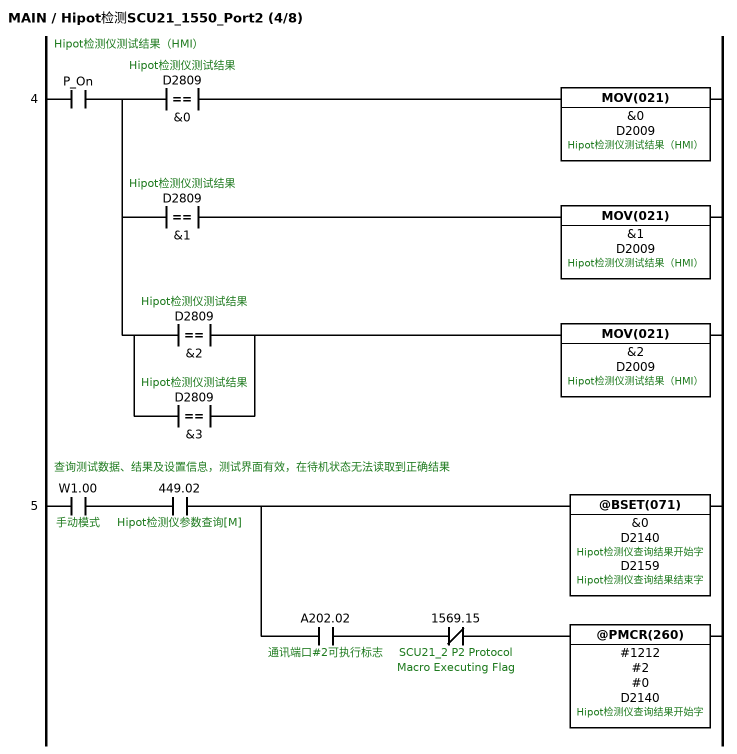
; [picture p48: MAIN / Hipot检测SCU21_1550_Port2, rungs 4-5]
; rung 4: Hipot检测仪测试结果（HMI）
LD P_On
OUT TR0
AND=(300) D2809 &0  ; Hipot检测仪测试结果
MOV(021) &0 D2009  ; Hipot检测仪测试结果（HMI）  // 0=无测试
LD TR0
AND=(300) D2809 &1  ; Hipot检测仪测试结果
MOV(021) &1 D2009  ; Hipot检测仪测试结果（HMI）  // 1=OK
LD TR0
LD=(300) D2809 &2  ; Hipot检测仪测试结果
OR=(300) D2809 &3  ; Hipot检测仪测试结果
ANDLD
MOV(021) &2 D2009  ; Hipot检测仪测试结果（HMI）  // 2=NG
; rung 5: 查询测试数据、结果及设置信息，测试界面有效，在待机状态无法读取到正确结果
LD W1.00  ; 手动模式
AND 449.02  ; Hipot检测仪参数查询[M]
@BSET(071) &0 D2140 D2159  ; Hipot检测仪查询结果开始字, Hipot检测仪查询结果结束字
AND A202.02  ; 通讯端口#2可执行标志
ANDNOT 1569.15  ; SCU21_2 P2 Protocol Macro Executing Flag
@PMCR(260) #1212 #2 #0 D2140  ; Hipot检测仪查询结果开始字

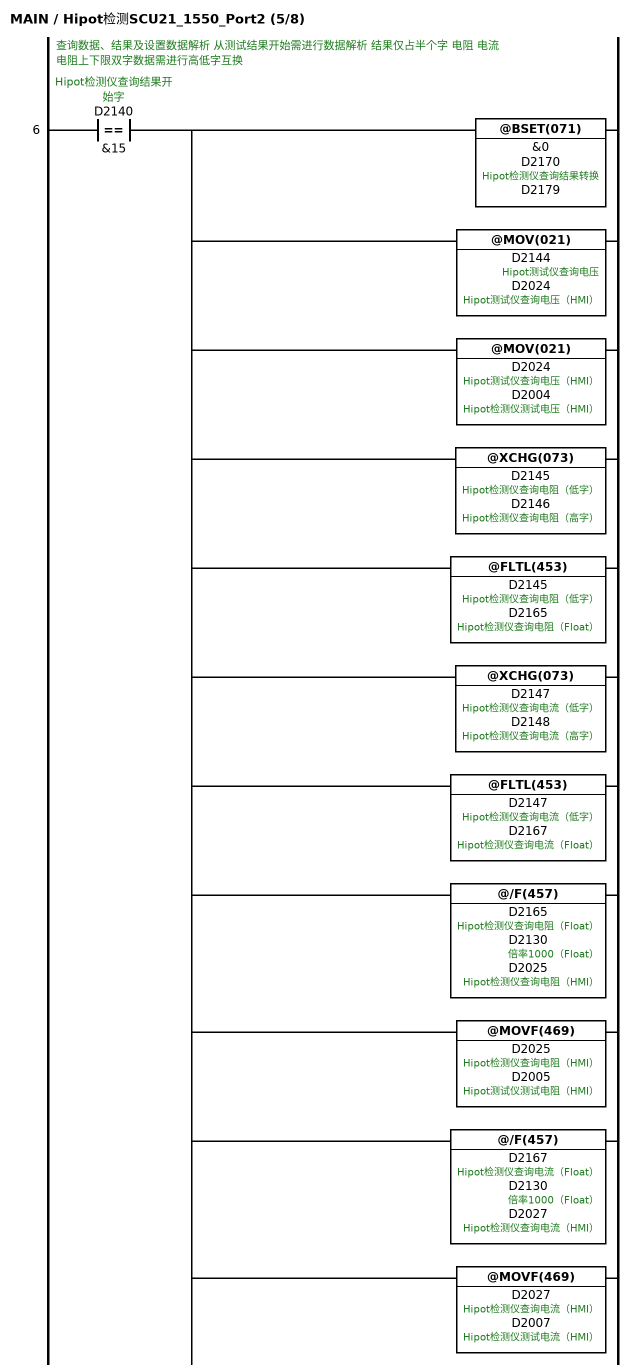

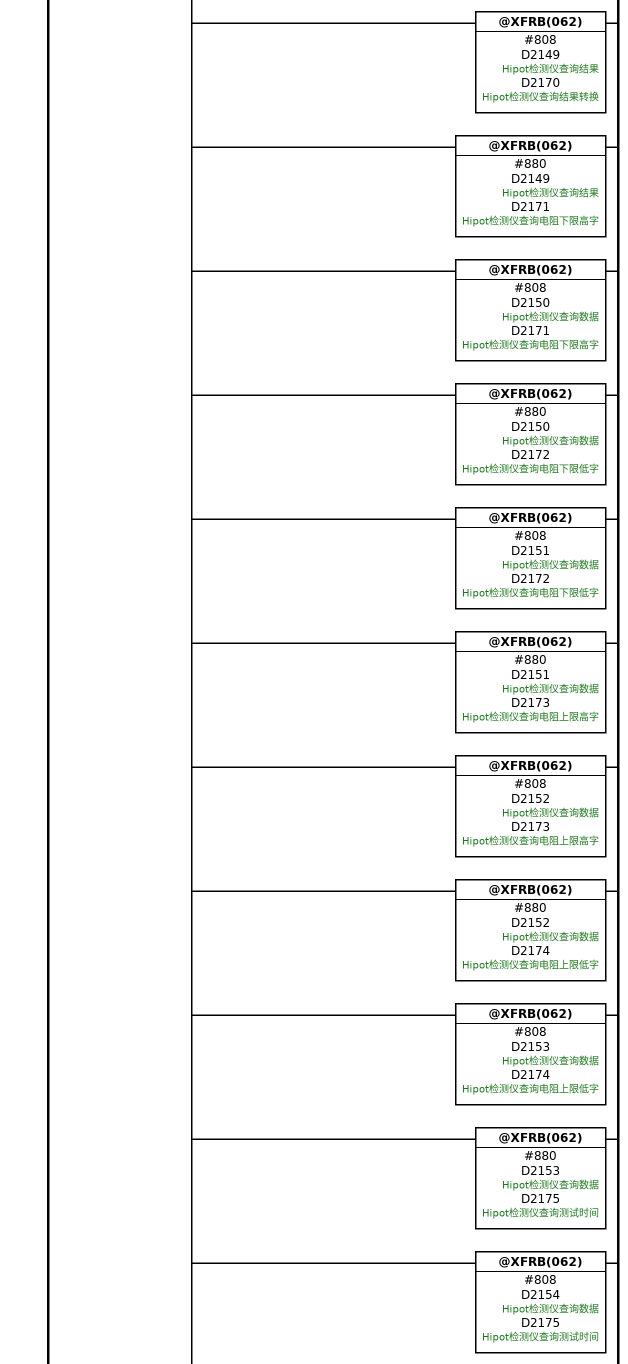

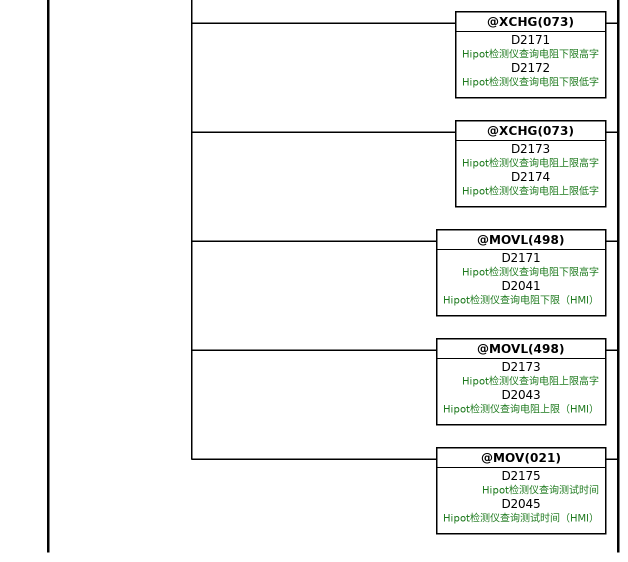
; rung 6: 查询数据、结果及设置数据解析 从测试结果开始需进行数据解析 结果仅占半个字 电阻 电流 电阻上下限双字数据需进行高低字互换
LD=(300) D2140 &15  ; Hipot检测仪查询结果开始字
@BSET(071) &0 D2170 D2179  ; Hipot检测仪查询结果转换
@MOV(021) D2144 D2024  ; Hipot测试仪查询电压, Hipot测试仪查询电压（HMI）
@MOV(021) D2024 D2004  ; Hipot测试仪查询电压（HMI）, Hipot检测仪测试电压（HMI）
@XCHG(073) D2145 D2146  ; Hipot检测仪查询电阻（低字）, Hipot检测仪查询电阻（高字）
@FLTL(453) D2145 D2165  ; Hipot检测仪查询电阻（低字）, Hipot检测仪查询电阻（Float）
@XCHG(073) D2147 D2148  ; Hipot检测仪查询电流（低字）, Hipot检测仪查询电流（高字）
@FLTL(453) D2147 D2167  ; Hipot检测仪查询电流（低字）, Hipot检测仪查询电流（Float）
@/F(457) D2165 D2130 D2025  ; Hipot检测仪查询电阻（Float）, 倍率1000（Float）, Hipot检测仪查询电阻（HMI）  // KΩ→MΩ
@MOVF(469) D2025 D2005  ; Hipot检测仪查询电阻（HMI）, Hipot测试仪测试电阻（HMI）
@/F(457) D2167 D2130 D2027  ; Hipot检测仪查询电流（Float）, 倍率1000（Float）, Hipot检测仪查询电流（HMI）  // nA→uA
@MOVF(469) D2027 D2007  ; Hipot检测仪查询电流（HMI）, Hipot检测仪测试电流（HMI）
@XFRB(062) #808 D2149 D2170  ; Hipot检测仪查询结果, Hipot检测仪查询结果转换
@XFRB(062) #880 D2149 D2171  ; Hipot检测仪查询结果, Hipot检测仪查询电阻下限高字
@XFRB(062) #808 D2150 D2171  ; Hipot检测仪查询数据, Hipot检测仪查询电阻下限高字
@XFRB(062) #880 D2150 D2172  ; Hipot检测仪查询数据, Hipot检测仪查询电阻下限低字
@XFRB(062) #808 D2151 D2172  ; Hipot检测仪查询数据, Hipot检测仪查询电阻下限低字
@XFRB(062) #880 D2151 D2173  ; Hipot检测仪查询数据, Hipot检测仪查询电阻上限高字
@XFRB(062) #808 D2152 D2173  ; Hipot检测仪查询数据, Hipot检测仪查询电阻上限高字
@XFRB(062) #880 D2152 D2174  ; Hipot检测仪查询数据, Hipot检测仪查询电阻上限低字
@XFRB(062) #808 D2153 D2174  ; Hipot检测仪查询数据, Hipot检测仪查询电阻上限低字
@XFRB(062) #880 D2153 D2175  ; Hipot检测仪查询数据, Hipot检测仪查询测试时间
@XFRB(062) #808 D2154 D2175  ; Hipot检测仪查询数据, Hipot检测仪查询测试时间
@XCHG(073) D2171 D2172  ; Hipot检测仪查询电阻下限高字, Hipot检测仪查询电阻下限低字
@XCHG(073) D2173 D2174  ; Hipot检测仪查询电阻上限高字, Hipot检测仪查询电阻上限低字
@MOVL(498) D2171 D2041  ; Hipot检测仪查询电阻下限高字, Hipot检测仪查询电阻下限（HMI）
@MOVL(498) D2173 D2043  ; Hipot检测仪查询电阻上限高字, Hipot检测仪查询电阻上限（HMI）
@MOV(021) D2175 D2045  ; Hipot检测仪查询测试时间, Hipot检测仪查询测试时间（HMI）

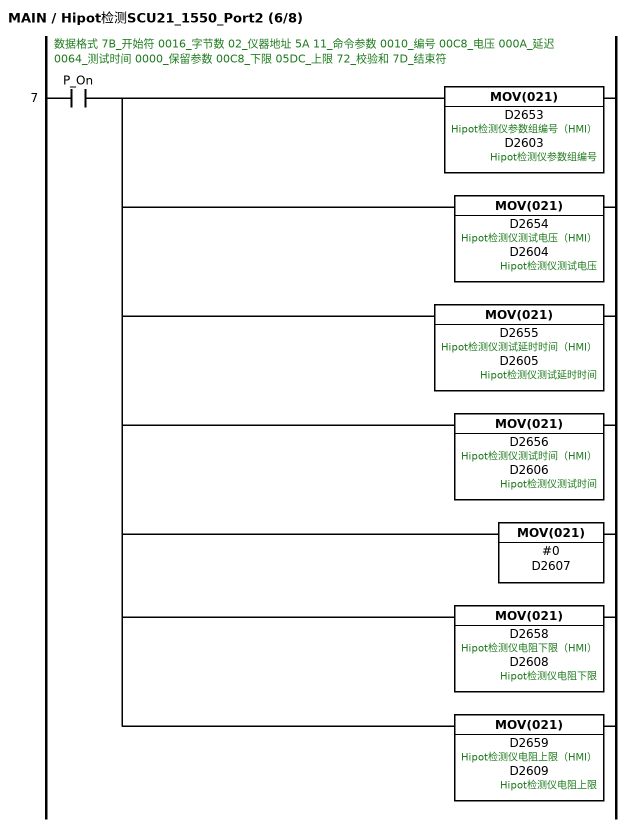
; rung 7: 数据格式 7B_开始符 0016_字节数 02_仪器地址 5A 11_命令参数 0010_编号 00C8_电压 000A_延迟 0064_测试时间 0000_保留参数 00C8_下限 05DC_上限 72_校验和 7D_结束符
LD P_On
MOV(021) D2653 D2603  ; Hipot检测仪参数组编号（HMI）, Hipot检测仪参数组编号
MOV(021) D2654 D2604  ; Hipot检测仪测试电压（HMI）, Hipot检测仪测试电压
MOV(021) D2655 D2605  ; Hipot检测仪测试延时时间（HMI）, Hipot检测仪测试延时时间
MOV(021) D2656 D2606  ; Hipot检测仪测试时间（HMI）, Hipot检测仪测试时间
MOV(021) #0 D2607
MOV(021) D2658 D2608  ; Hipot检测仪电阻下限（HMI）, Hipot检测仪电阻下限
MOV(021) D2659 D2609  ; Hipot检测仪电阻上限（HMI）, Hipot检测仪电阻上限

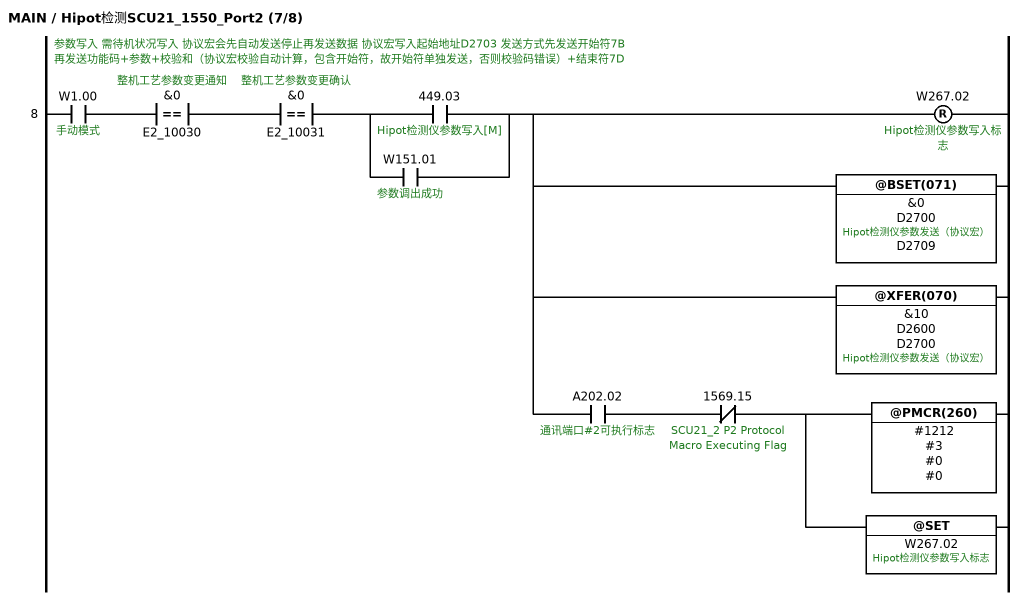
; rung 8: 参数写入 需待机状况写入 协议宏会先自动发送停止再发送数据 协议宏写入起始地址D2703 发送方式先发送开始符7B 再发送功能码+参数+校验和（协议宏校验自动计算，包含开始符，故开始符单独发送，否则校验码错误）+结束符7D
LD W1.00  ; 手动模式
AND=(300) &0 E2_10030  ; 整机工艺参数变更通知
AND=(300) &0 E2_10031  ; 整机工艺参数变更确认
LD 449.03  ; Hipot检测仪参数写入[M]
OR W151.01  ; 参数调出成功
ANDLD
RSET W267.02  ; Hipot检测仪参数写入标志
@BSET(071) &0 D2700 D2709  ; Hipot检测仪参数发送（协议宏）
@XFER(070) &10 D2600 D2700  ; Hipot检测仪参数发送（协议宏）
AND A202.02  ; 通讯端口#2可执行标志
ANDNOT 1569.15  ; SCU21_2 P2 Protocol Macro Executing Flag
@PMCR(260) #1212 #3 #0 #0
@SET W267.02  ; Hipot检测仪参数写入标志

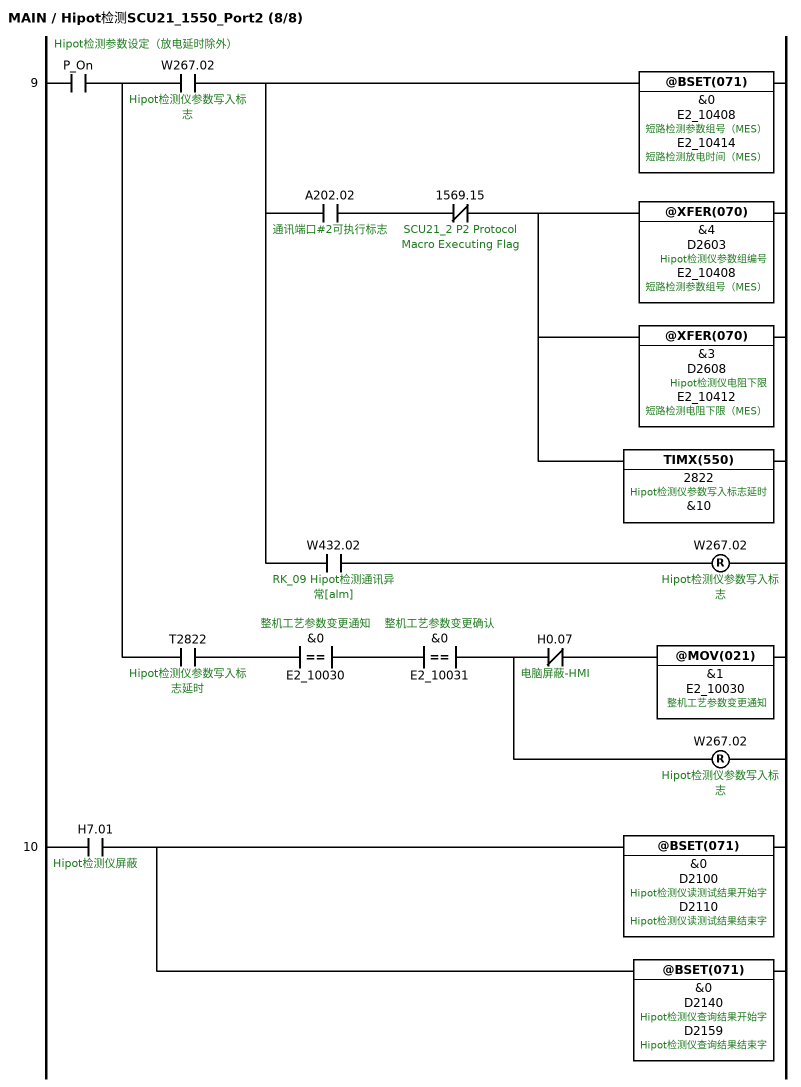
; rung 9: Hipot检测参数设定（放电延时除外）
LD P_On
OUT TR0
AND W267.02  ; Hipot检测仪参数写入标志
OUT TR1
@BSET(071) &0 E2_10408 E2_10414  ; 短路检测参数组号（MES）, 短路检测放电时间（MES）
AND A202.02  ; 通讯端口#2可执行标志
ANDNOT 1569.15  ; SCU21_2 P2 Protocol Macro Executing Flag
@XFER(070) &4 D2603 E2_10408  ; Hipot检测仪参数组编号, 短路检测参数组号（MES）
@XFER(070) &3 D2608 E2_10412  ; Hipot检测仪电阻下限, 短路检测电阻下限（MES）
TIMX(550) 2822 &10  ; Hipot检测仪参数写入标志延时
LD TR1
AND W432.02  ; RK_09 Hipot检测通讯异常[alm]
RSET W267.02  ; Hipot检测仪参数写入标志
LD TR0
AND T2822  ; Hipot检测仪参数写入标志延时
AND=(300) &0 E2_10030  ; 整机工艺参数变更通知
AND=(300) &0 E2_10031  ; 整机工艺参数变更确认
OUT TR0
ANDNOT H0.07  ; 电脑屏蔽-HMI
@MOV(021) &1 E2_10030  ; 整机工艺参数变更通知
LD TR0
RSET W267.02  ; Hipot检测仪参数写入标志
; rung 10
LD H7.01  ; Hipot检测仪屏蔽
@BSET(071) &0 D2100 D2110  ; Hipot检测仪读测试结果开始字, Hipot检测仪读测试结果结束字
@BSET(071) &0 D2140 D2159  ; Hipot检测仪查询结果开始字, Hipot检测仪查询结果结束字

### Section NC433_0_2000

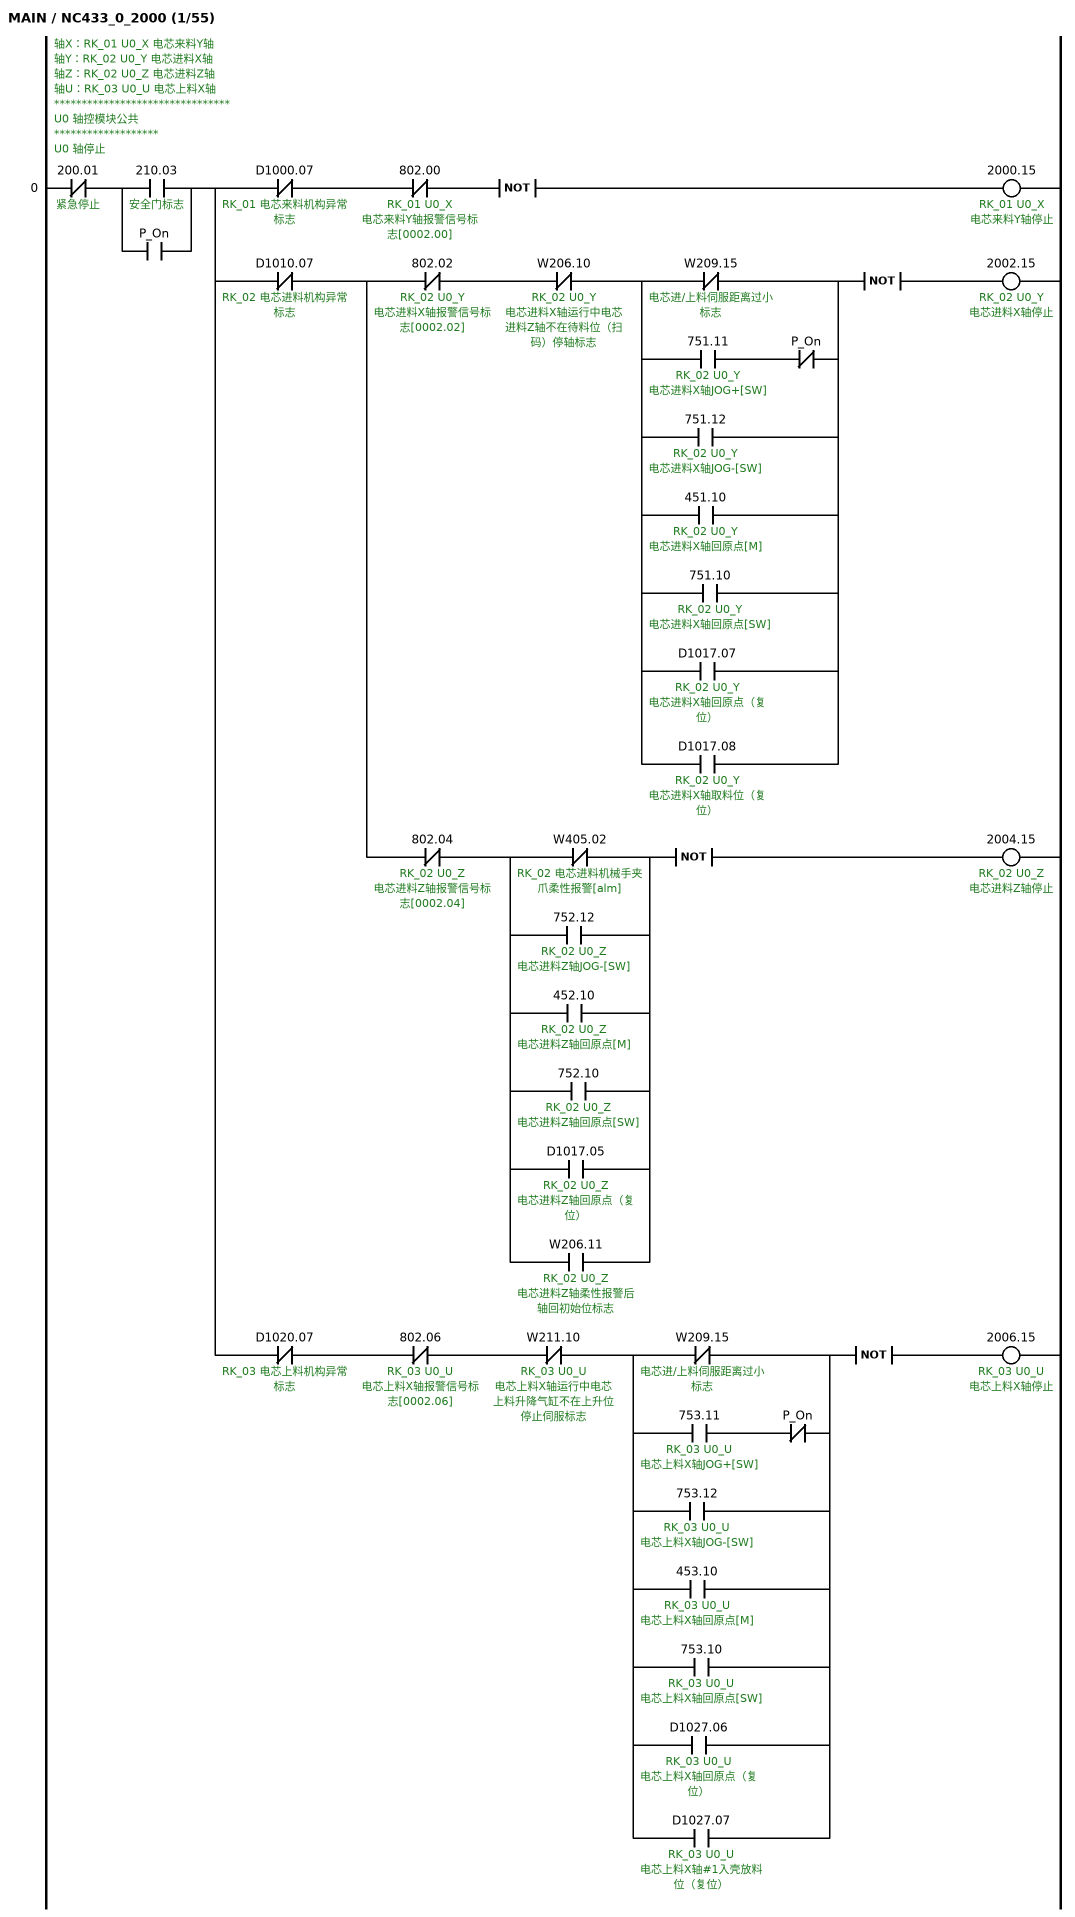
; rung 0: 轴X：RK_01 U0_X 电芯来料Y轴 / 轴Y：RK_02 U0_Y 电芯进料X轴 / 轴Z：RK_02 U0_Z 电芯进料Z轴 / 轴U：RK_03 U0_U 电芯上料X轴 / ******************************** / U0 轴控模块公共 / ******************* / U0 轴停止
LDNOT 200.01  ; 紧急停止
LD 210.03  ; 安全门标志
OR P_On
ANDLD
OUT TR0
ANDNOT D1000.07  ; RK_01 电芯来料机构异常标志
ANDNOT 802.00  ; RK_01 U0_X 电芯来料Y轴报警信号标志[0002.00]
NOT(520)
OUT 2000.15  ; RK_01 U0_X 电芯来料Y轴停止
LD TR0
ANDNOT D1010.07  ; RK_02 电芯进料机构异常标志
OUT TR1
ANDNOT 802.02  ; RK_02 U0_Y 电芯进料X轴报警信号标志[0002.02]
ANDNOT W206.10  ; RK_02 U0_Y 电芯进料X轴运行中电芯进料Z轴不在待料位（扫码）停轴标志
LDNOT W209.15  ; 电芯进/上料伺服距离过小标志
LD 751.11  ; RK_02 U0_Y 电芯进料X轴JOG+[SW]
ANDNOT P_On
ORLD
OR 751.12  ; RK_02 U0_Y 电芯进料X轴JOG-[SW]
OR 451.10  ; RK_02 U0_Y 电芯进料X轴回原点[M]
OR 751.10  ; RK_02 U0_Y 电芯进料X轴回原点[SW]
OR D1017.07  ; RK_02 U0_Y 电芯进料X轴回原点（复位）
OR D1017.08  ; RK_02 U0_Y 电芯进料X轴取料位（复位）
ANDLD
NOT(520)
OUT 2002.15  ; RK_02 U0_Y 电芯进料X轴停止
LD TR1
ANDNOT 802.04  ; RK_02 U0_Z 电芯进料Z轴报警信号标志[0002.04]
LDNOT W405.02  ; RK_02 电芯进料机械手夹爪柔性报警[alm]
OR 752.12  ; RK_02 U0_Z 电芯进料Z轴JOG-[SW]
OR 452.10  ; RK_02 U0_Z 电芯进料Z轴回原点[M]
OR 752.10  ; RK_02 U0_Z 电芯进料Z轴回原点[SW]
OR D1017.05  ; RK_02 U0_Z 电芯进料Z轴回原点（复位）
OR W206.11  ; RK_02 U0_Z 电芯进料Z轴柔性报警后轴回初始位标志
ANDLD
NOT(520)
OUT 2004.15  ; RK_02 U0_Z 电芯进料Z轴停止
LD TR0
ANDNOT D1020.07  ; RK_03 电芯上料机构异常标志
ANDNOT 802.06  ; RK_03 U0_U 电芯上料X轴报警信号标志[0002.06]
ANDNOT W211.10  ; RK_03 U0_U 电芯上料X轴运行中电芯上料升降气缸不在上升位停止伺服标志
LDNOT W209.15  ; 电芯进/上料伺服距离过小标志
LD 753.11  ; RK_03 U0_U 电芯上料X轴JOG+[SW]
ANDNOT P_On
ORLD
OR 753.12  ; RK_03 U0_U 电芯上料X轴JOG-[SW]
OR 453.10  ; RK_03 U0_U 电芯上料X轴回原点[M]
OR 753.10  ; RK_03 U0_U 电芯上料X轴回原点[SW]
OR D1027.06  ; RK_03 U0_U 电芯上料X轴回原点（复位）
OR D1027.07  ; RK_03 U0_U 电芯上料X轴#1入壳放料位（复位）
ANDLD
NOT(520)
OUT 2006.15  ; RK_03 U0_U 电芯上料X轴停止

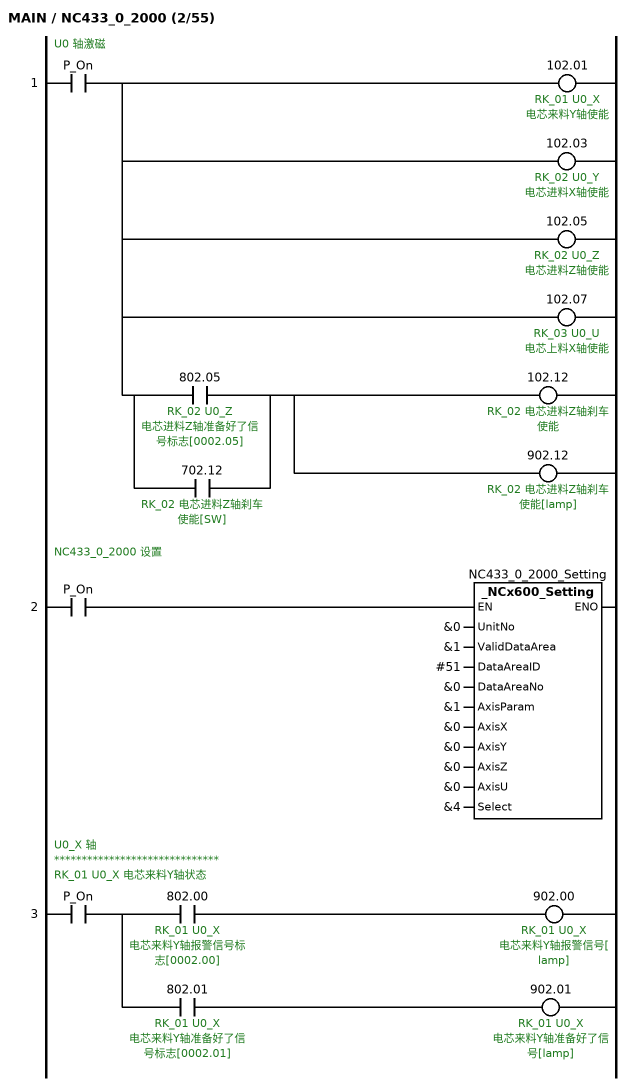
; rung 1: U0 轴激磁
LD P_On
OUT 102.01  ; RK_01 U0_X 电芯来料Y轴使能
OUT 102.03  ; RK_02 U0_Y 电芯进料X轴使能
OUT 102.05  ; RK_02 U0_Z 电芯进料Z轴使能
OUT 102.07  ; RK_03 U0_U 电芯上料X轴使能
LD 802.05  ; RK_02 U0_Z 电芯进料Z轴准备好了信号标志[0002.05]
OR 702.12  ; RK_02 电芯进料Z轴刹车使能[SW]
ANDLD
OUT 102.12  ; RK_02 电芯进料Z轴刹车使能
OUT 902.12  ; RK_02 电芯进料Z轴刹车使能[lamp]
; rung 2: NC433_0_2000 设置
LD P_On
CALL NC433_0_2000_Setting : _NCx600_Setting (UnitNo := &0, ValidDataArea := &1, DataAreaID := #51, DataAreaNo := &0, AxisParam := &1, AxisX := &0, AxisY := &0, AxisZ := &0, AxisU := &0, Select := &4)
; rung 3: U0_X 轴 / ****************************** / RK_01 U0_X 电芯来料Y轴状态
LD P_On
OUT TR0
AND 802.00  ; RK_01 U0_X 电芯来料Y轴报警信号标志[0002.00]
OUT 902.00  ; RK_01 U0_X 电芯来料Y轴报警信号[lamp]
LD TR0
AND 802.01  ; RK_01 U0_X 电芯来料Y轴准备好了信号标志[0002.01]
OUT 902.01  ; RK_01 U0_X 电芯来料Y轴准备好了信号[lamp]

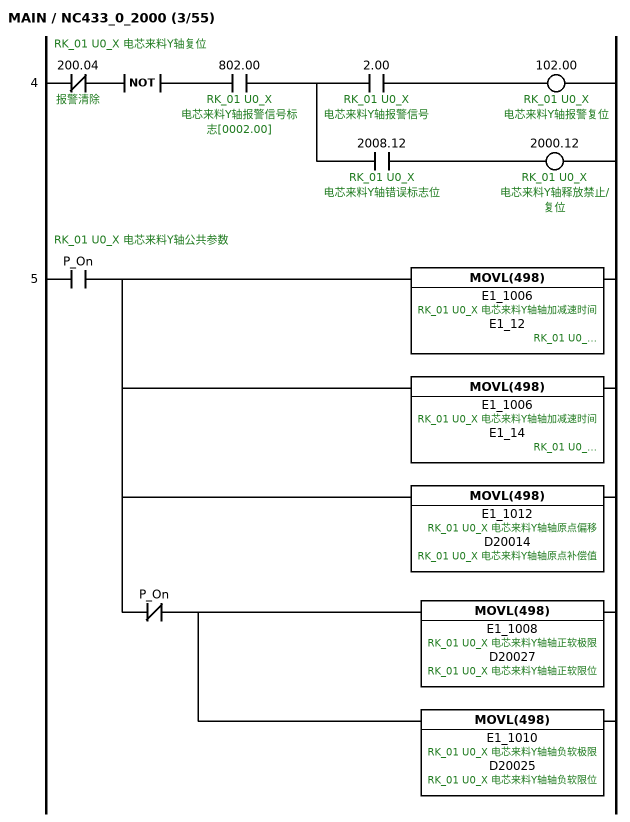
; rung 4: RK_01 U0_X 电芯来料Y轴复位
LDNOT 200.04  ; 报警清除
NOT(520)
AND 802.00  ; RK_01 U0_X 电芯来料Y轴报警信号标志[0002.00]
OUT TR0
AND 2.00  ; RK_01 U0_X 电芯来料Y轴报警信号
OUT 102.00  ; RK_01 U0_X 电芯来料Y轴报警复位
LD TR0
AND 2008.12  ; RK_01 U0_X 电芯来料Y轴错误标志位
OUT 2000.12  ; RK_01 U0_X 电芯来料Y轴释放禁止/复位
; rung 5: RK_01 U0_X 电芯来料Y轴公共参数
LD P_On
MOVL(498) E1_1006 E1_12  ; RK_01 U0_X 电芯来料Y轴轴加减速时间, RK_01 U0_X 电芯来料Y轴轴直接操作加速时间
MOVL(498) E1_1006 E1_14  ; RK_01 U0_X 电芯来料Y轴轴加减速时间, RK_01 U0_X 电芯来料Y轴轴直接操作减速时间
MOVL(498) E1_1012 D20014  ; RK_01 U0_X 电芯来料Y轴轴原点偏移, RK_01 U0_X 电芯来料Y轴轴原点补偿值
ANDNOT P_On
MOVL(498) E1_1008 D20027  ; RK_01 U0_X 电芯来料Y轴轴正软极限, RK_01 U0_X 电芯来料Y轴轴正软限位
MOVL(498) E1_1010 D20025  ; RK_01 U0_X 电芯来料Y轴轴负软极限, RK_01 U0_X 电芯来料Y轴轴负软限位

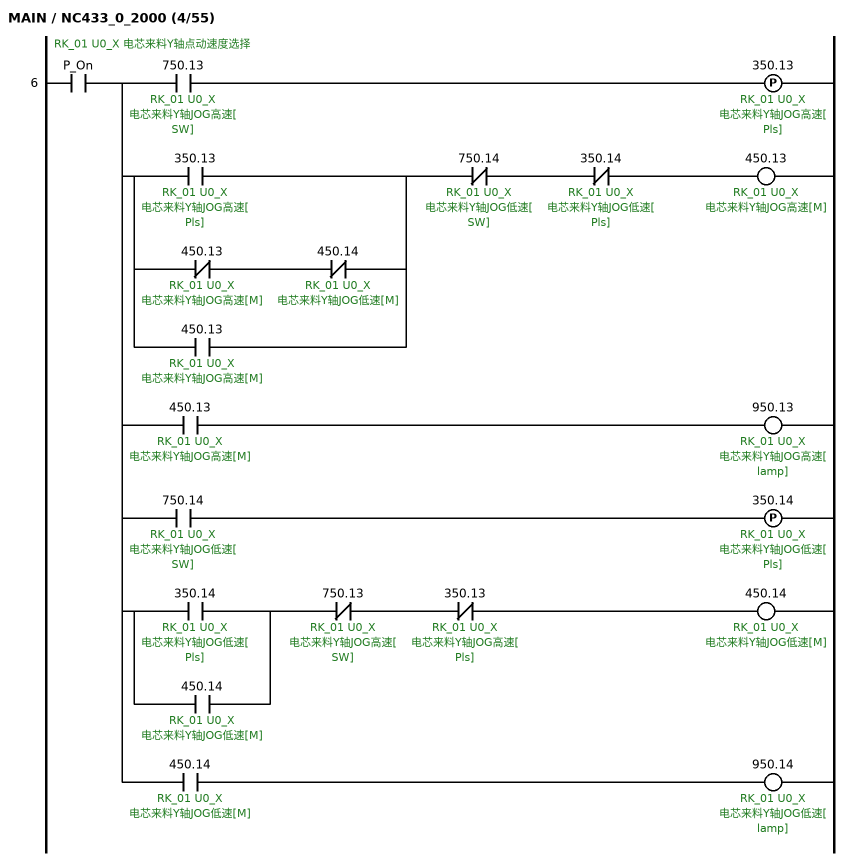
; rung 6: RK_01 U0_X 电芯来料Y轴点动速度选择
LD P_On
OUT TR0
AND 750.13  ; RK_01 U0_X 电芯来料Y轴JOG高速[SW]
DIFU(013) 350.13  ; RK_01 U0_X 电芯来料Y轴JOG高速[Pls]
LD TR0
LD 350.13  ; RK_01 U0_X 电芯来料Y轴JOG高速[Pls]
LDNOT 450.13  ; RK_01 U0_X 电芯来料Y轴JOG高速[M]
ANDNOT 450.14  ; RK_01 U0_X 电芯来料Y轴JOG低速[M]
ORLD
OR 450.13  ; RK_01 U0_X 电芯来料Y轴JOG高速[M]
ANDLD
ANDNOT 750.14  ; RK_01 U0_X 电芯来料Y轴JOG低速[SW]
ANDNOT 350.14  ; RK_01 U0_X 电芯来料Y轴JOG低速[Pls]
OUT 450.13  ; RK_01 U0_X 电芯来料Y轴JOG高速[M]
LD TR0
AND 450.13  ; RK_01 U0_X 电芯来料Y轴JOG高速[M]
OUT 950.13  ; RK_01 U0_X 电芯来料Y轴JOG高速[lamp]
LD TR0
AND 750.14  ; RK_01 U0_X 电芯来料Y轴JOG低速[SW]
DIFU(013) 350.14  ; RK_01 U0_X 电芯来料Y轴JOG低速[Pls]
LD TR0
LD 350.14  ; RK_01 U0_X 电芯来料Y轴JOG低速[Pls]
OR 450.14  ; RK_01 U0_X 电芯来料Y轴JOG低速[M]
ANDLD
ANDNOT 750.13  ; RK_01 U0_X 电芯来料Y轴JOG高速[SW]
ANDNOT 350.13  ; RK_01 U0_X 电芯来料Y轴JOG高速[Pls]
OUT 450.14  ; RK_01 U0_X 电芯来料Y轴JOG低速[M]
LD TR0
AND 450.14  ; RK_01 U0_X 电芯来料Y轴JOG低速[M]
OUT 950.14  ; RK_01 U0_X 电芯来料Y轴JOG低速[lamp]

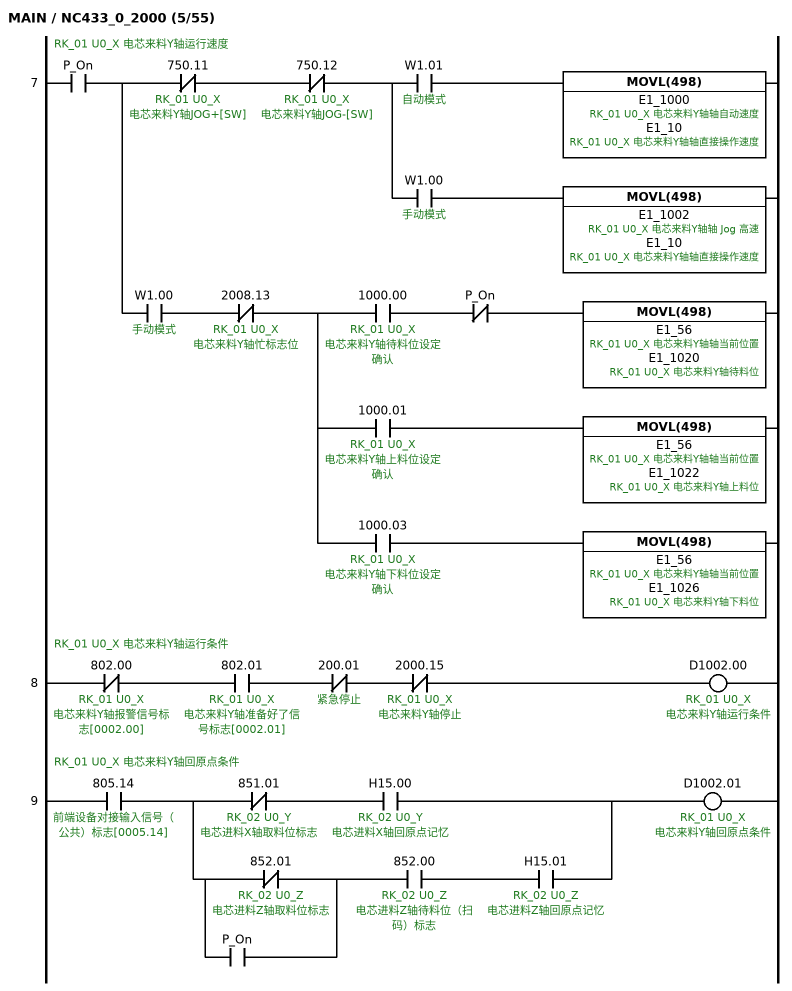
; rung 7: RK_01 U0_X 电芯来料Y轴运行速度
LD P_On
OUT TR0
ANDNOT 750.11  ; RK_01 U0_X 电芯来料Y轴JOG+[SW]
ANDNOT 750.12  ; RK_01 U0_X 电芯来料Y轴JOG-[SW]
OUT TR1
AND W1.01  ; 自动模式
MOVL(498) E1_1000 E1_10  ; RK_01 U0_X 电芯来料Y轴轴自动速度, RK_01 U0_X 电芯来料Y轴轴直接操作速度
LD TR1
AND W1.00  ; 手动模式
MOVL(498) E1_1002 E1_10  ; RK_01 U0_X 电芯来料Y轴轴 Jog 高速, RK_01 U0_X 电芯来料Y轴轴直接操作速度
LD TR0
AND W1.00  ; 手动模式
ANDNOT 2008.13  ; RK_01 U0_X 电芯来料Y轴忙标志位
OUT TR0
AND 1000.00  ; RK_01 U0_X 电芯来料Y轴待料位设定确认
ANDNOT P_On
MOVL(498) E1_56 E1_1020  ; RK_01 U0_X 电芯来料Y轴轴当前位置, RK_01 U0_X 电芯来料Y轴待料位
LD TR0
AND 1000.01  ; RK_01 U0_X 电芯来料Y轴上料位设定确认
MOVL(498) E1_56 E1_1022  ; RK_01 U0_X 电芯来料Y轴轴当前位置, RK_01 U0_X 电芯来料Y轴上料位
LD TR0
AND 1000.03  ; RK_01 U0_X 电芯来料Y轴下料位设定确认
MOVL(498) E1_56 E1_1026  ; RK_01 U0_X 电芯来料Y轴轴当前位置, RK_01 U0_X 电芯来料Y轴下料位
; rung 8: RK_01 U0_X 电芯来料Y轴运行条件
LDNOT 802.00  ; RK_01 U0_X 电芯来料Y轴报警信号标志[0002.00]
AND 802.01  ; RK_01 U0_X 电芯来料Y轴准备好了信号标志[0002.01]
ANDNOT 200.01  ; 紧急停止
ANDNOT 2000.15  ; RK_01 U0_X 电芯来料Y轴停止
OUT D1002.00  ; RK_01 U0_X 电芯来料Y轴运行条件
; rung 9: RK_01 U0_X 电芯来料Y轴回原点条件
LD 805.14  ; 前端设备对接输入信号（公共）标志[0005.14]  // 前端设备放料中（放料中=1）！！
LDNOT 851.01  ; RK_02 U0_Y 电芯进料X轴取料位标志  // 严格来讲应该设定：设定大值XXXX<电芯进料X轴<设定小值XXXX
AND H15.00  ; RK_02 U0_Y 电芯进料X轴回原点记忆
LDNOT 852.01  ; RK_02 U0_Z 电芯进料Z轴取料位标志
OR P_On
AND 852.00  ; RK_02 U0_Z 电芯进料Z轴待料位（扫码）标志
AND H15.01  ; RK_02 U0_Z 电芯进料Z轴回原点记忆
ORLD
ANDLD
OUT D1002.01  ; RK_01 U0_X 电芯来料Y轴回原点条件

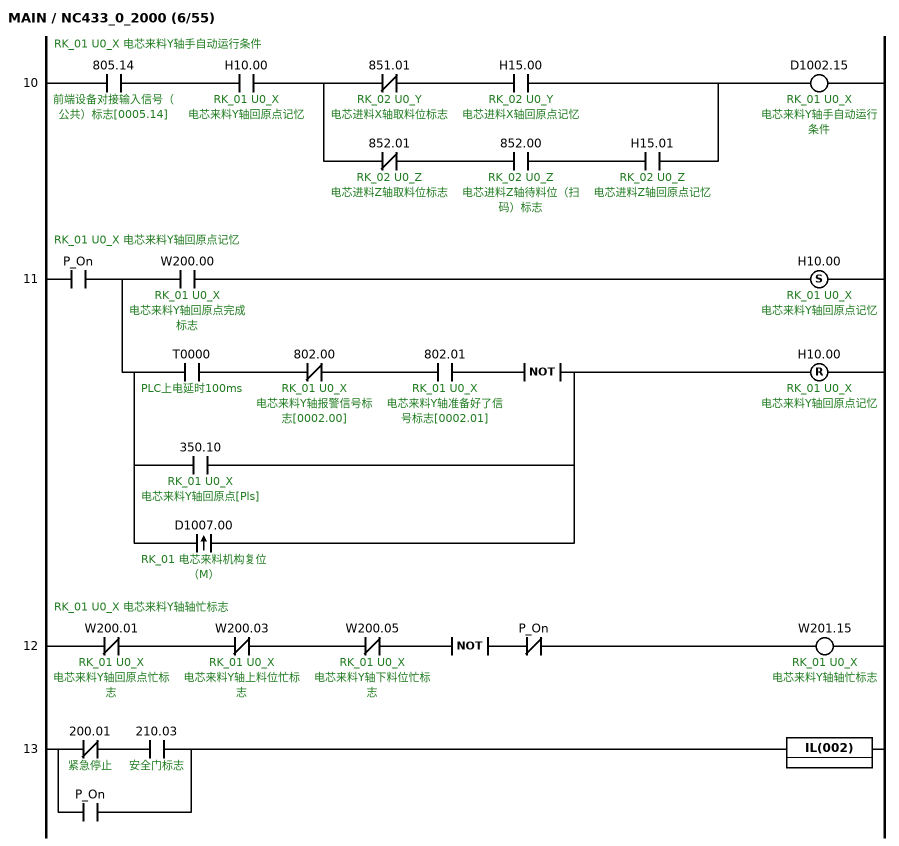
; rung 10: RK_01 U0_X 电芯来料Y轴手自动运行条件
LD 805.14  ; 前端设备对接输入信号（公共）标志[0005.14]  // 前端设备放料中（放料中=1）！
AND H10.00  ; RK_01 U0_X 电芯来料Y轴回原点记忆
LDNOT 851.01  ; RK_02 U0_Y 电芯进料X轴取料位标志
AND H15.00  ; RK_02 U0_Y 电芯进料X轴回原点记忆
LDNOT 852.01  ; RK_02 U0_Z 电芯进料Z轴取料位标志
AND 852.00  ; RK_02 U0_Z 电芯进料Z轴待料位（扫码）标志
AND H15.01  ; RK_02 U0_Z 电芯进料Z轴回原点记忆
ORLD
ANDLD
OUT D1002.15  ; RK_01 U0_X 电芯来料Y轴手自动运行条件
; rung 11: RK_01 U0_X 电芯来料Y轴回原点记忆
LD P_On
OUT TR0
AND W200.00  ; RK_01 U0_X 电芯来料Y轴回原点完成标志
SET H10.00  ; RK_01 U0_X 电芯来料Y轴回原点记忆
LD TR0
LD T0000  ; PLC上电延时100ms
ANDNOT 802.00  ; RK_01 U0_X 电芯来料Y轴报警信号标志[0002.00]
AND 802.01  ; RK_01 U0_X 电芯来料Y轴准备好了信号标志[0002.01]
NOT(520)
OR 350.10  ; RK_01 U0_X 电芯来料Y轴回原点[Pls]
@OR D1007.00  ; RK_01 电芯来料机构复位（M）
ANDLD
RSET H10.00  ; RK_01 U0_X 电芯来料Y轴回原点记忆
; rung 12: RK_01 U0_X 电芯来料Y轴轴忙标志
LDNOT W200.01  ; RK_01 U0_X 电芯来料Y轴回原点忙标志
ANDNOT W200.03  ; RK_01 U0_X 电芯来料Y轴上料位忙标志
ANDNOT W200.05  ; RK_01 U0_X 电芯来料Y轴下料位忙标志
NOT(520)
ANDNOT P_On
OUT W201.15  ; RK_01 U0_X 电芯来料Y轴轴忙标志
; rung 13
LDNOT 200.01  ; 紧急停止
AND 210.03  ; 安全门标志
OR P_On
IL(002)

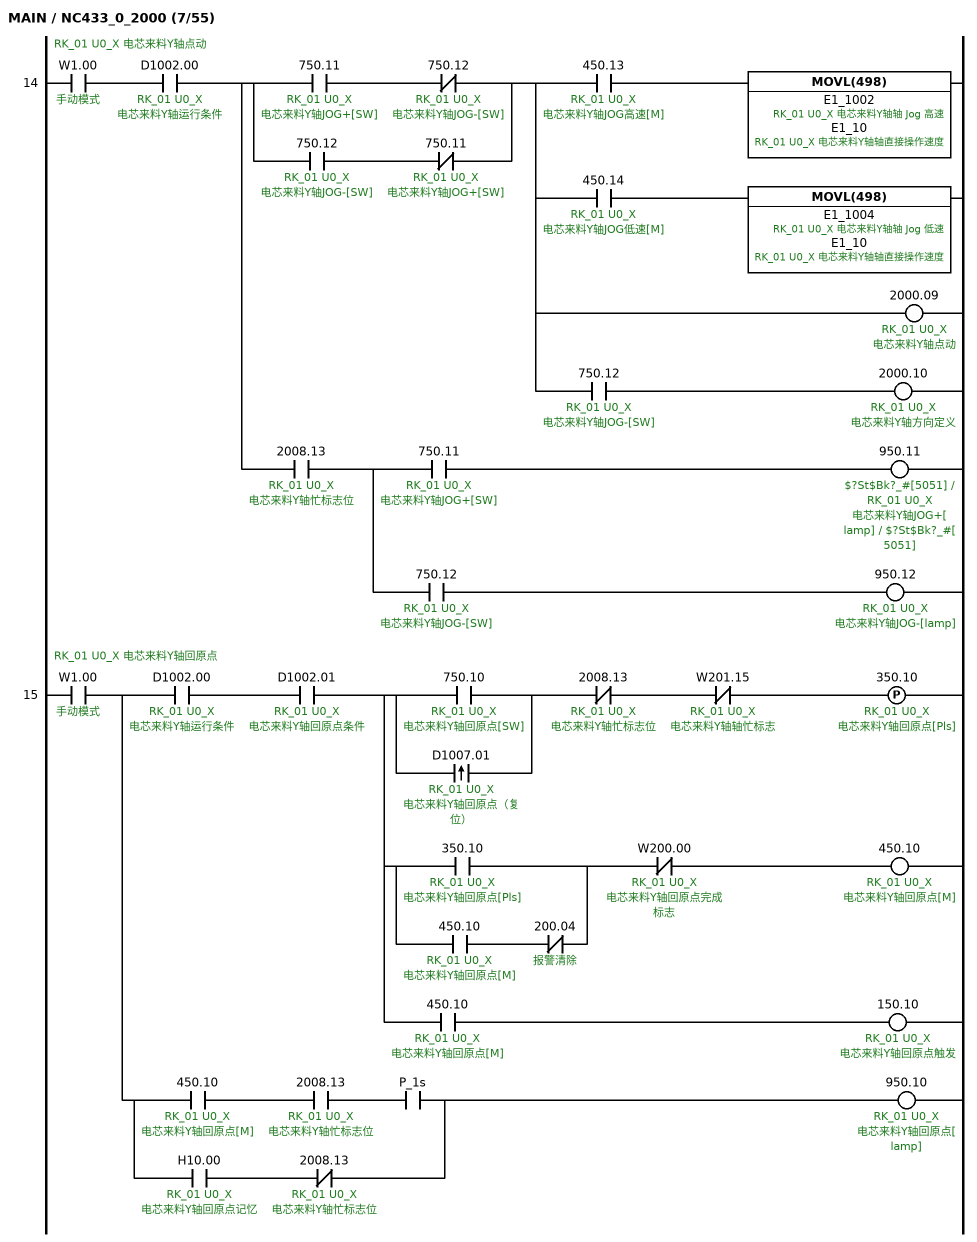
; rung 14: RK_01 U0_X 电芯来料Y轴点动
LD W1.00  ; 手动模式
AND D1002.00  ; RK_01 U0_X 电芯来料Y轴运行条件
OUT TR0
LD 750.11  ; RK_01 U0_X 电芯来料Y轴JOG+[SW]
ANDNOT 750.12  ; RK_01 U0_X 电芯来料Y轴JOG-[SW]
LD 750.12  ; RK_01 U0_X 电芯来料Y轴JOG-[SW]
ANDNOT 750.11  ; RK_01 U0_X 电芯来料Y轴JOG+[SW]
ORLD
ANDLD
OUT TR1
AND 450.13  ; RK_01 U0_X 电芯来料Y轴JOG高速[M]
MOVL(498) E1_1002 E1_10  ; RK_01 U0_X 电芯来料Y轴轴 Jog 高速, RK_01 U0_X 电芯来料Y轴轴直接操作速度
LD TR1
AND 450.14  ; RK_01 U0_X 电芯来料Y轴JOG低速[M]
MOVL(498) E1_1004 E1_10  ; RK_01 U0_X 电芯来料Y轴轴 Jog 低速, RK_01 U0_X 电芯来料Y轴轴直接操作速度
LD TR1
OUT 2000.09  ; RK_01 U0_X 电芯来料Y轴点动
AND 750.12  ; RK_01 U0_X 电芯来料Y轴JOG-[SW]
OUT 2000.10  ; RK_01 U0_X 电芯来料Y轴方向定义
LD TR0
AND 2008.13  ; RK_01 U0_X 电芯来料Y轴忙标志位
OUT TR0
AND 750.11  ; RK_01 U0_X 电芯来料Y轴JOG+[SW]
OUT 950.11  ; $?St$Bk?_#[5051] / RK_01 U0_X 电芯来料Y轴JOG+[lamp] / $?St$Bk?_#[5051]
LD TR0
AND 750.12  ; RK_01 U0_X 电芯来料Y轴JOG-[SW]
OUT 950.12  ; RK_01 U0_X 电芯来料Y轴JOG-[lamp]
; rung 15: RK_01 U0_X 电芯来料Y轴回原点
LD W1.00  ; 手动模式
OUT TR0
AND D1002.00  ; RK_01 U0_X 电芯来料Y轴运行条件
AND D1002.01  ; RK_01 U0_X 电芯来料Y轴回原点条件
OUT TR1
LD 750.10  ; RK_01 U0_X 电芯来料Y轴回原点[SW]
@OR D1007.01  ; RK_01 U0_X 电芯来料Y轴回原点（复位）
ANDLD
ANDNOT 2008.13  ; RK_01 U0_X 电芯来料Y轴忙标志位
ANDNOT W201.15  ; RK_01 U0_X 电芯来料Y轴轴忙标志
DIFU(013) 350.10  ; RK_01 U0_X 电芯来料Y轴回原点[Pls]
LD TR1
LD 350.10  ; RK_01 U0_X 电芯来料Y轴回原点[Pls]
LD 450.10  ; RK_01 U0_X 电芯来料Y轴回原点[M]
ANDNOT 200.04  ; 报警清除
ORLD
ANDLD
ANDNOT W200.00  ; RK_01 U0_X 电芯来料Y轴回原点完成标志
OUT 450.10  ; RK_01 U0_X 电芯来料Y轴回原点[M]
LD TR1
AND 450.10  ; RK_01 U0_X 电芯来料Y轴回原点[M]
OUT 150.10  ; RK_01 U0_X 电芯来料Y轴回原点触发
LD TR0
LD 450.10  ; RK_01 U0_X 电芯来料Y轴回原点[M]
AND 2008.13  ; RK_01 U0_X 电芯来料Y轴忙标志位
AND P_1s
LD H10.00  ; RK_01 U0_X 电芯来料Y轴回原点记忆
ANDNOT 2008.13  ; RK_01 U0_X 电芯来料Y轴忙标志位
ORLD
ANDLD
OUT 950.10  ; RK_01 U0_X 电芯来料Y轴回原点[lamp]

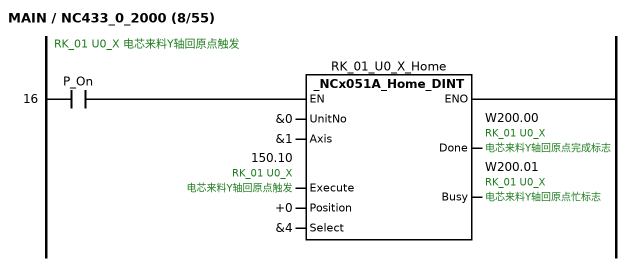
; rung 16: RK_01 U0_X 电芯来料Y轴回原点触发
LD P_On
CALL RK_01_U0_X_Home : _NCx051A_Home_DINT (UnitNo := &0, Axis := &1, Execute := 150.10, Position := +0, Select := &4, Done => W200.00, Busy => W200.01)  ; RK_01 U0_X 电芯来料Y轴回原点触发, RK_01 U0_X 电芯来料Y轴回原点完成标志, RK_01 U0_X 电芯来料Y轴回原点忙标志

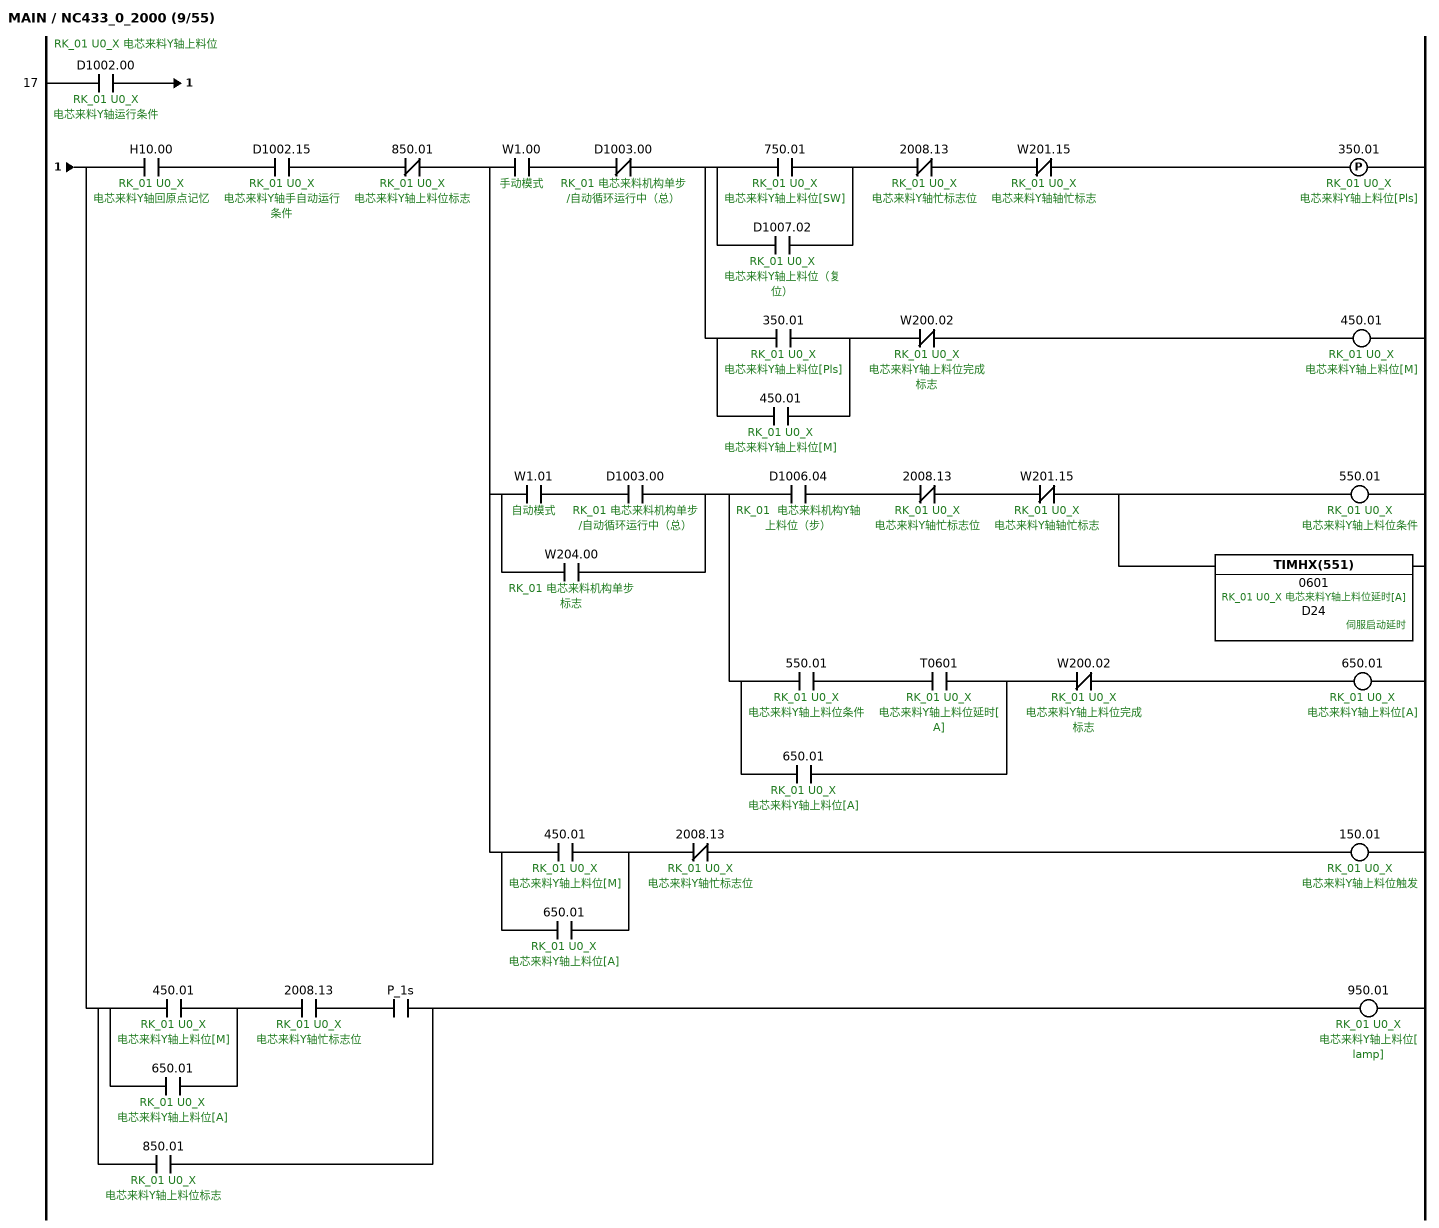
; rung 17: RK_01 U0_X 电芯来料Y轴上料位
LD D1002.00  ; RK_01 U0_X 电芯来料Y轴运行条件
OUT TR0
AND H10.00  ; RK_01 U0_X 电芯来料Y轴回原点记忆
AND D1002.15  ; RK_01 U0_X 电芯来料Y轴手自动运行条件
ANDNOT 850.01  ; RK_01 U0_X 电芯来料Y轴上料位标志
OUT TR1
AND W1.00  ; 手动模式
ANDNOT D1003.00  ; RK_01 电芯来料机构单步/自动循环运行中（总）
OUT TR2
LD 750.01  ; RK_01 U0_X 电芯来料Y轴上料位[SW]
OR D1007.02  ; RK_01 U0_X 电芯来料Y轴上料位（复位）
ANDLD
ANDNOT 2008.13  ; RK_01 U0_X 电芯来料Y轴忙标志位
ANDNOT W201.15  ; RK_01 U0_X 电芯来料Y轴轴忙标志
DIFU(013) 350.01  ; RK_01 U0_X 电芯来料Y轴上料位[Pls]
LD TR2
LD 350.01  ; RK_01 U0_X 电芯来料Y轴上料位[Pls]
OR 450.01  ; RK_01 U0_X 电芯来料Y轴上料位[M]
ANDLD
ANDNOT W200.02  ; RK_01 U0_X 电芯来料Y轴上料位完成标志
OUT 450.01  ; RK_01 U0_X 电芯来料Y轴上料位[M]
LD TR1
LD W1.01  ; 自动模式
AND D1003.00  ; RK_01 电芯来料机构单步/自动循环运行中（总）
OR W204.00  ; RK_01 电芯来料机构单步标志
ANDLD
OUT TR2
AND D1006.04  ; RK_01  电芯来料机构Y轴上料位（步）
ANDNOT 2008.13  ; RK_01 U0_X 电芯来料Y轴忙标志位
ANDNOT W201.15  ; RK_01 U0_X 电芯来料Y轴轴忙标志
OUT 550.01  ; RK_01 U0_X 电芯来料Y轴上料位条件
TIMHX(551) 0601 D24  ; 伺服启动延时, RK_01 U0_X 电芯来料Y轴上料位延时[A]
LD TR2
LD 550.01  ; RK_01 U0_X 电芯来料Y轴上料位条件
AND T0601  ; RK_01 U0_X 电芯来料Y轴上料位延时[A]
OR 650.01  ; RK_01 U0_X 电芯来料Y轴上料位[A]
ANDLD
ANDNOT W200.02  ; RK_01 U0_X 电芯来料Y轴上料位完成标志
OUT 650.01  ; RK_01 U0_X 电芯来料Y轴上料位[A]
LD TR1
LD 450.01  ; RK_01 U0_X 电芯来料Y轴上料位[M]
OR 650.01  ; RK_01 U0_X 电芯来料Y轴上料位[A]
ANDLD
ANDNOT 2008.13  ; RK_01 U0_X 电芯来料Y轴忙标志位
OUT 150.01  ; RK_01 U0_X 电芯来料Y轴上料位触发
LD TR0
LD 450.01  ; RK_01 U0_X 电芯来料Y轴上料位[M]
OR 650.01  ; RK_01 U0_X 电芯来料Y轴上料位[A]
AND 2008.13  ; RK_01 U0_X 电芯来料Y轴忙标志位
AND P_1s
OR 850.01  ; RK_01 U0_X 电芯来料Y轴上料位标志
ANDLD
OUT 950.01  ; RK_01 U0_X 电芯来料Y轴上料位[lamp]

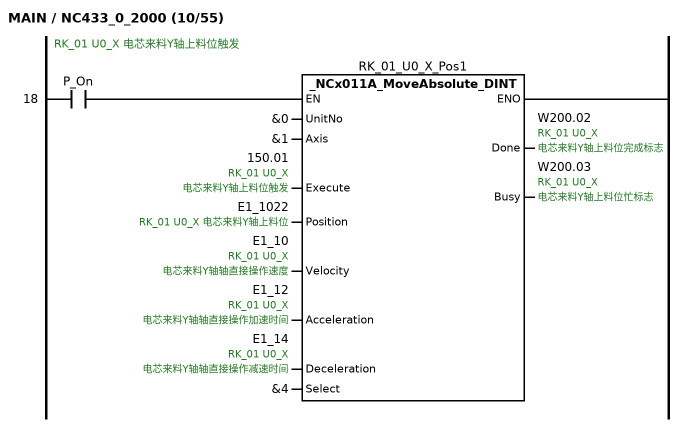
; rung 18: RK_01 U0_X 电芯来料Y轴上料位触发
LD P_On
CALL RK_01_U0_X_Pos1 : _NCx011A_MoveAbsolute_DINT (UnitNo := &0, Axis := &1, Execute := 150.01, Position := E1_1022, Velocity := E1_10, Acceleration := E1_12, Deceleration := E1_14, Select := &4, Done => W200.02, Busy => W200.03)  ; RK_01 U0_X 电芯来料Y轴上料位触发, RK_01 U0_X 电芯来料Y轴上料位, RK_01 U0_X 电芯来料Y轴轴直接操作速度, RK_01 U0_X 电芯来料Y轴轴直接操作加速时间, RK_01 U0_X 电芯来料Y轴轴直接操作减速时间, RK_01 U0_X 电芯来料Y轴上料位完成标志, RK_01 U0_X 电芯来料Y轴上料位忙标志

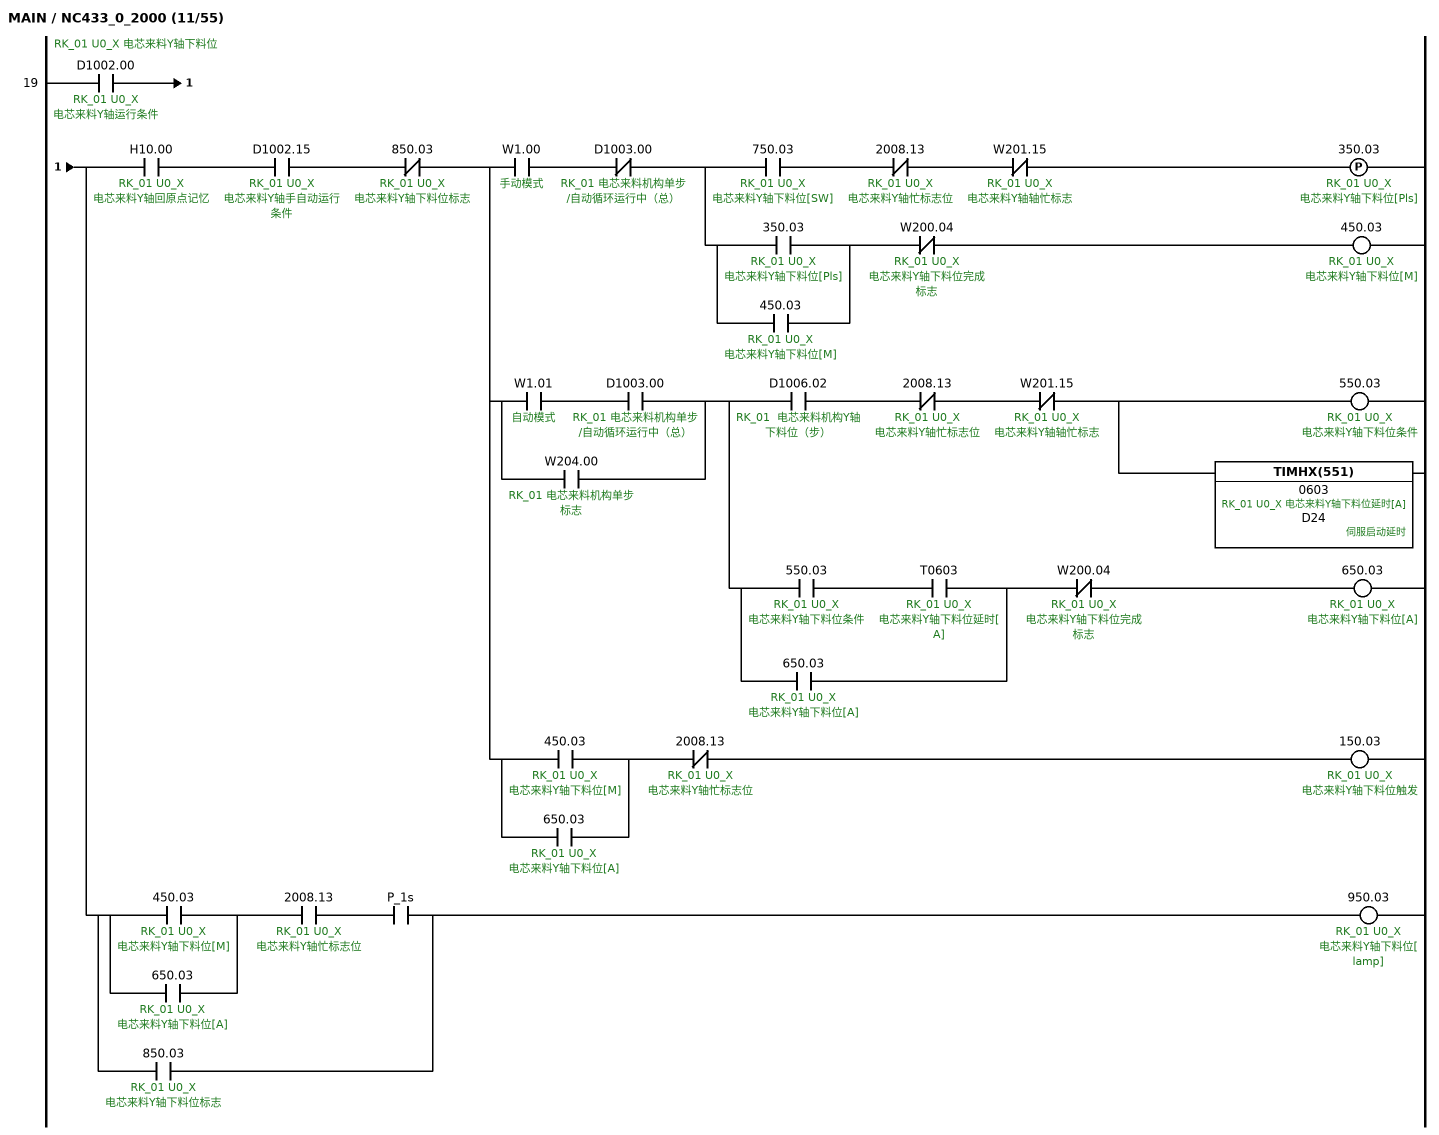
; rung 19: RK_01 U0_X 电芯来料Y轴下料位
LD D1002.00  ; RK_01 U0_X 电芯来料Y轴运行条件
OUT TR0
AND H10.00  ; RK_01 U0_X 电芯来料Y轴回原点记忆
AND D1002.15  ; RK_01 U0_X 电芯来料Y轴手自动运行条件
ANDNOT 850.03  ; RK_01 U0_X 电芯来料Y轴下料位标志
OUT TR1
AND W1.00  ; 手动模式
ANDNOT D1003.00  ; RK_01 电芯来料机构单步/自动循环运行中（总）
OUT TR2
AND 750.03  ; RK_01 U0_X 电芯来料Y轴下料位[SW]
ANDNOT 2008.13  ; RK_01 U0_X 电芯来料Y轴忙标志位
ANDNOT W201.15  ; RK_01 U0_X 电芯来料Y轴轴忙标志
DIFU(013) 350.03  ; RK_01 U0_X 电芯来料Y轴下料位[Pls]
LD TR2
LD 350.03  ; RK_01 U0_X 电芯来料Y轴下料位[Pls]
OR 450.03  ; RK_01 U0_X 电芯来料Y轴下料位[M]
ANDLD
ANDNOT W200.04  ; RK_01 U0_X 电芯来料Y轴下料位完成标志
OUT 450.03  ; RK_01 U0_X 电芯来料Y轴下料位[M]
LD TR1
LD W1.01  ; 自动模式
AND D1003.00  ; RK_01 电芯来料机构单步/自动循环运行中（总）
OR W204.00  ; RK_01 电芯来料机构单步标志
ANDLD
OUT TR2
AND D1006.02  ; RK_01  电芯来料机构Y轴下料位（步）
ANDNOT 2008.13  ; RK_01 U0_X 电芯来料Y轴忙标志位
ANDNOT W201.15  ; RK_01 U0_X 电芯来料Y轴轴忙标志
OUT 550.03  ; RK_01 U0_X 电芯来料Y轴下料位条件
TIMHX(551) 0603 D24  ; 伺服启动延时, RK_01 U0_X 电芯来料Y轴下料位延时[A]
LD TR2
LD 550.03  ; RK_01 U0_X 电芯来料Y轴下料位条件
AND T0603  ; RK_01 U0_X 电芯来料Y轴下料位延时[A]
OR 650.03  ; RK_01 U0_X 电芯来料Y轴下料位[A]
ANDLD
ANDNOT W200.04  ; RK_01 U0_X 电芯来料Y轴下料位完成标志
OUT 650.03  ; RK_01 U0_X 电芯来料Y轴下料位[A]
LD TR1
LD 450.03  ; RK_01 U0_X 电芯来料Y轴下料位[M]
OR 650.03  ; RK_01 U0_X 电芯来料Y轴下料位[A]
ANDLD
ANDNOT 2008.13  ; RK_01 U0_X 电芯来料Y轴忙标志位
OUT 150.03  ; RK_01 U0_X 电芯来料Y轴下料位触发
LD TR0
LD 450.03  ; RK_01 U0_X 电芯来料Y轴下料位[M]
OR 650.03  ; RK_01 U0_X 电芯来料Y轴下料位[A]
AND 2008.13  ; RK_01 U0_X 电芯来料Y轴忙标志位
AND P_1s
OR 850.03  ; RK_01 U0_X 电芯来料Y轴下料位标志
ANDLD
OUT 950.03  ; RK_01 U0_X 电芯来料Y轴下料位[lamp]

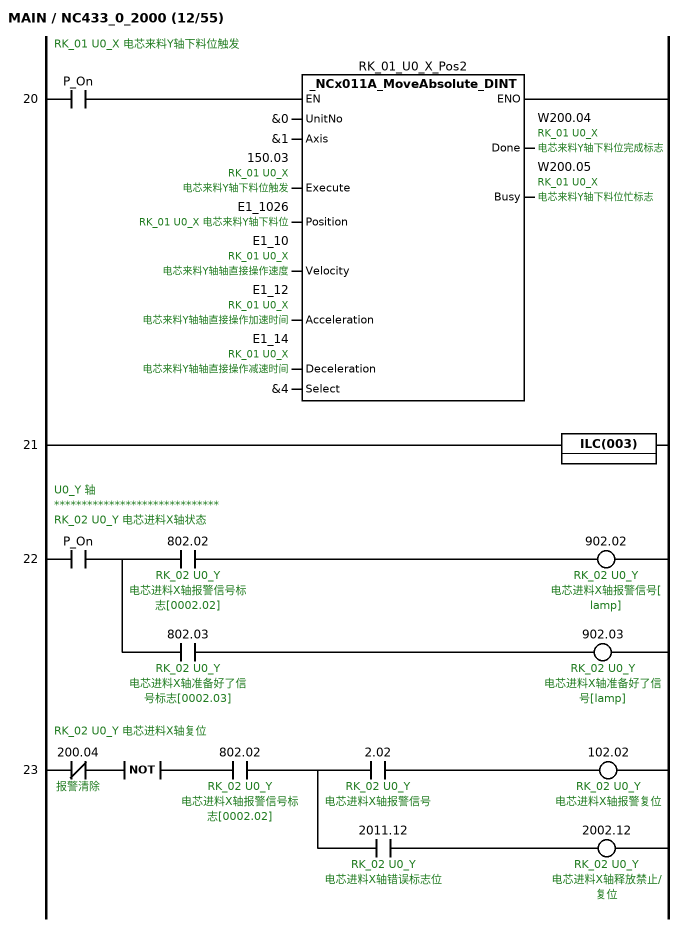
; rung 20: RK_01 U0_X 电芯来料Y轴下料位触发
LD P_On
CALL RK_01_U0_X_Pos2 : _NCx011A_MoveAbsolute_DINT (UnitNo := &0, Axis := &1, Execute := 150.03, Position := E1_1026, Velocity := E1_10, Acceleration := E1_12, Deceleration := E1_14, Select := &4, Done => W200.04, Busy => W200.05)  ; RK_01 U0_X 电芯来料Y轴下料位触发, RK_01 U0_X 电芯来料Y轴下料位, RK_01 U0_X 电芯来料Y轴轴直接操作速度, RK_01 U0_X 电芯来料Y轴轴直接操作加速时间, RK_01 U0_X 电芯来料Y轴轴直接操作减速时间, RK_01 U0_X 电芯来料Y轴下料位完成标志, RK_01 U0_X 电芯来料Y轴下料位忙标志
; rung 21
ILC(003)
; rung 22: U0_Y 轴 / ****************************** / RK_02 U0_Y 电芯进料X轴状态
LD P_On
OUT TR0
AND 802.02  ; RK_02 U0_Y 电芯进料X轴报警信号标志[0002.02]
OUT 902.02  ; RK_02 U0_Y 电芯进料X轴报警信号[lamp]
LD TR0
AND 802.03  ; RK_02 U0_Y 电芯进料X轴准备好了信号标志[0002.03]
OUT 902.03  ; RK_02 U0_Y 电芯进料X轴准备好了信号[lamp]
; rung 23: RK_02 U0_Y 电芯进料X轴复位
LDNOT 200.04  ; 报警清除
NOT(520)
AND 802.02  ; RK_02 U0_Y 电芯进料X轴报警信号标志[0002.02]
OUT TR0
AND 2.02  ; RK_02 U0_Y 电芯进料X轴报警信号
OUT 102.02  ; RK_02 U0_Y 电芯进料X轴报警复位
LD TR0
AND 2011.12  ; RK_02 U0_Y 电芯进料X轴错误标志位
OUT 2002.12  ; RK_02 U0_Y 电芯进料X轴释放禁止/复位

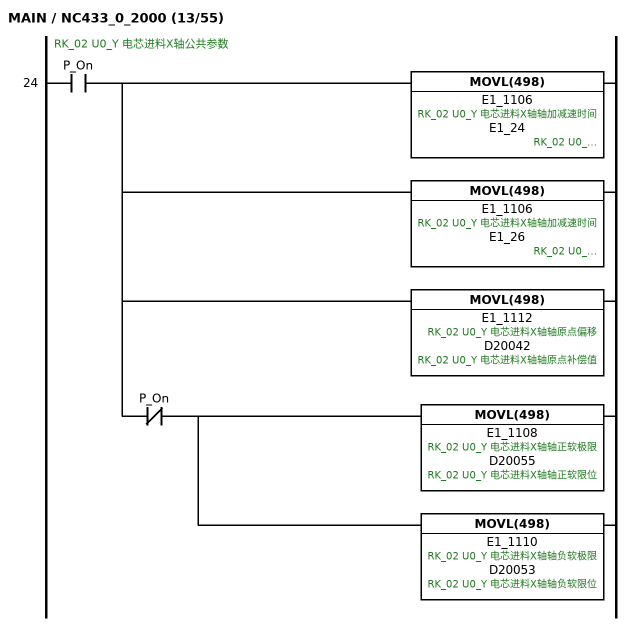
; rung 24: RK_02 U0_Y 电芯进料X轴公共参数
LD P_On
MOVL(498) E1_1106 E1_24  ; RK_02 U0_Y 电芯进料X轴轴加减速时间, RK_02 U0_Y 电芯进料X轴轴直接操作加速时间
MOVL(498) E1_1106 E1_26  ; RK_02 U0_Y 电芯进料X轴轴加减速时间, RK_02 U0_Y 电芯进料X轴轴直接操作减速时间
MOVL(498) E1_1112 D20042  ; RK_02 U0_Y 电芯进料X轴轴原点偏移, RK_02 U0_Y 电芯进料X轴轴原点补偿值
ANDNOT P_On
MOVL(498) E1_1108 D20055  ; RK_02 U0_Y 电芯进料X轴轴正软极限, RK_02 U0_Y 电芯进料X轴轴正软限位
MOVL(498) E1_1110 D20053  ; RK_02 U0_Y 电芯进料X轴轴负软极限, RK_02 U0_Y 电芯进料X轴轴负软限位

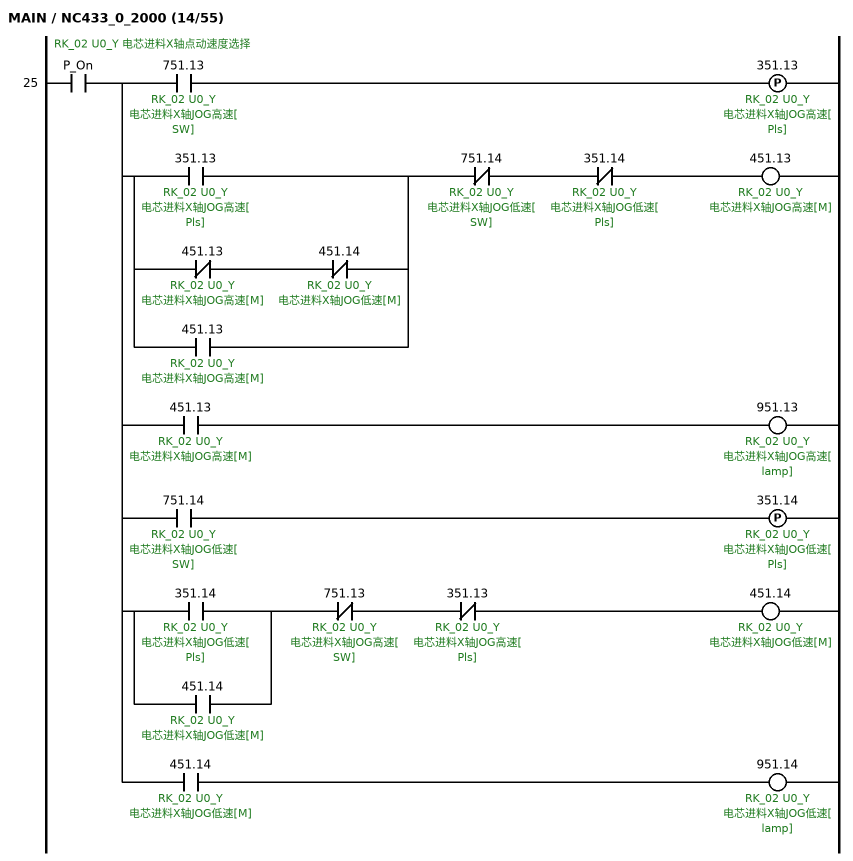
; rung 25: RK_02 U0_Y 电芯进料X轴点动速度选择
LD P_On
OUT TR0
AND 751.13  ; RK_02 U0_Y 电芯进料X轴JOG高速[SW]
DIFU(013) 351.13  ; RK_02 U0_Y 电芯进料X轴JOG高速[Pls]
LD TR0
LD 351.13  ; RK_02 U0_Y 电芯进料X轴JOG高速[Pls]
LDNOT 451.13  ; RK_02 U0_Y 电芯进料X轴JOG高速[M]
ANDNOT 451.14  ; RK_02 U0_Y 电芯进料X轴JOG低速[M]
ORLD
OR 451.13  ; RK_02 U0_Y 电芯进料X轴JOG高速[M]
ANDLD
ANDNOT 751.14  ; RK_02 U0_Y 电芯进料X轴JOG低速[SW]
ANDNOT 351.14  ; RK_02 U0_Y 电芯进料X轴JOG低速[Pls]
OUT 451.13  ; RK_02 U0_Y 电芯进料X轴JOG高速[M]
LD TR0
AND 451.13  ; RK_02 U0_Y 电芯进料X轴JOG高速[M]
OUT 951.13  ; RK_02 U0_Y 电芯进料X轴JOG高速[lamp]
LD TR0
AND 751.14  ; RK_02 U0_Y 电芯进料X轴JOG低速[SW]
DIFU(013) 351.14  ; RK_02 U0_Y 电芯进料X轴JOG低速[Pls]
LD TR0
LD 351.14  ; RK_02 U0_Y 电芯进料X轴JOG低速[Pls]
OR 451.14  ; RK_02 U0_Y 电芯进料X轴JOG低速[M]
ANDLD
ANDNOT 751.13  ; RK_02 U0_Y 电芯进料X轴JOG高速[SW]
ANDNOT 351.13  ; RK_02 U0_Y 电芯进料X轴JOG高速[Pls]
OUT 451.14  ; RK_02 U0_Y 电芯进料X轴JOG低速[M]
LD TR0
AND 451.14  ; RK_02 U0_Y 电芯进料X轴JOG低速[M]
OUT 951.14  ; RK_02 U0_Y 电芯进料X轴JOG低速[lamp]

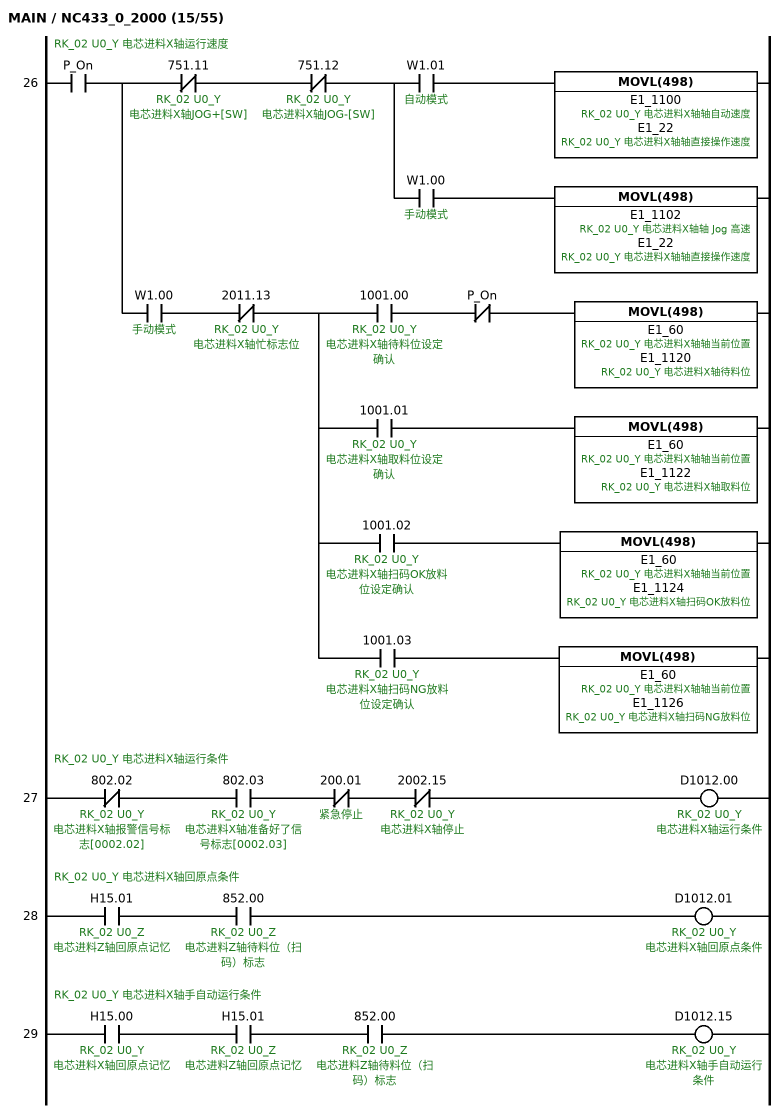
; rung 26: RK_02 U0_Y 电芯进料X轴运行速度
LD P_On
OUT TR0
ANDNOT 751.11  ; RK_02 U0_Y 电芯进料X轴JOG+[SW]
ANDNOT 751.12  ; RK_02 U0_Y 电芯进料X轴JOG-[SW]
OUT TR1
AND W1.01  ; 自动模式
MOVL(498) E1_1100 E1_22  ; RK_02 U0_Y 电芯进料X轴轴自动速度, RK_02 U0_Y 电芯进料X轴轴直接操作速度
LD TR1
AND W1.00  ; 手动模式
MOVL(498) E1_1102 E1_22  ; RK_02 U0_Y 电芯进料X轴轴 Jog 高速, RK_02 U0_Y 电芯进料X轴轴直接操作速度
LD TR0
AND W1.00  ; 手动模式
ANDNOT 2011.13  ; RK_02 U0_Y 电芯进料X轴忙标志位
OUT TR0
AND 1001.00  ; RK_02 U0_Y 电芯进料X轴待料位设定确认
ANDNOT P_On
MOVL(498) E1_60 E1_1120  ; RK_02 U0_Y 电芯进料X轴轴当前位置, RK_02 U0_Y 电芯进料X轴待料位
LD TR0
AND 1001.01  ; RK_02 U0_Y 电芯进料X轴取料位设定确认
MOVL(498) E1_60 E1_1122  ; RK_02 U0_Y 电芯进料X轴轴当前位置, RK_02 U0_Y 电芯进料X轴取料位
LD TR0
AND 1001.02  ; RK_02 U0_Y 电芯进料X轴扫码OK放料位设定确认
MOVL(498) E1_60 E1_1124  ; RK_02 U0_Y 电芯进料X轴轴当前位置, RK_02 U0_Y 电芯进料X轴扫码OK放料位
LD TR0
AND 1001.03  ; RK_02 U0_Y 电芯进料X轴扫码NG放料位设定确认
MOVL(498) E1_60 E1_1126  ; RK_02 U0_Y 电芯进料X轴轴当前位置, RK_02 U0_Y 电芯进料X轴扫码NG放料位
; rung 27: RK_02 U0_Y 电芯进料X轴运行条件
LDNOT 802.02  ; RK_02 U0_Y 电芯进料X轴报警信号标志[0002.02]
AND 802.03  ; RK_02 U0_Y 电芯进料X轴准备好了信号标志[0002.03]
ANDNOT 200.01  ; 紧急停止
ANDNOT 2002.15  ; RK_02 U0_Y 电芯进料X轴停止
OUT D1012.00  ; RK_02 U0_Y 电芯进料X轴运行条件
; rung 28: RK_02 U0_Y 电芯进料X轴回原点条件
LD H15.01  ; RK_02 U0_Z 电芯进料Z轴回原点记忆
AND 852.00  ; RK_02 U0_Z 电芯进料Z轴待料位（扫码）标志
OUT D1012.01  ; RK_02 U0_Y 电芯进料X轴回原点条件
; rung 29: RK_02 U0_Y 电芯进料X轴手自动运行条件
LD H15.00  ; RK_02 U0_Y 电芯进料X轴回原点记忆
AND H15.01  ; RK_02 U0_Z 电芯进料Z轴回原点记忆
AND 852.00  ; RK_02 U0_Z 电芯进料Z轴待料位（扫码）标志
OUT D1012.15  ; RK_02 U0_Y 电芯进料X轴手自动运行条件

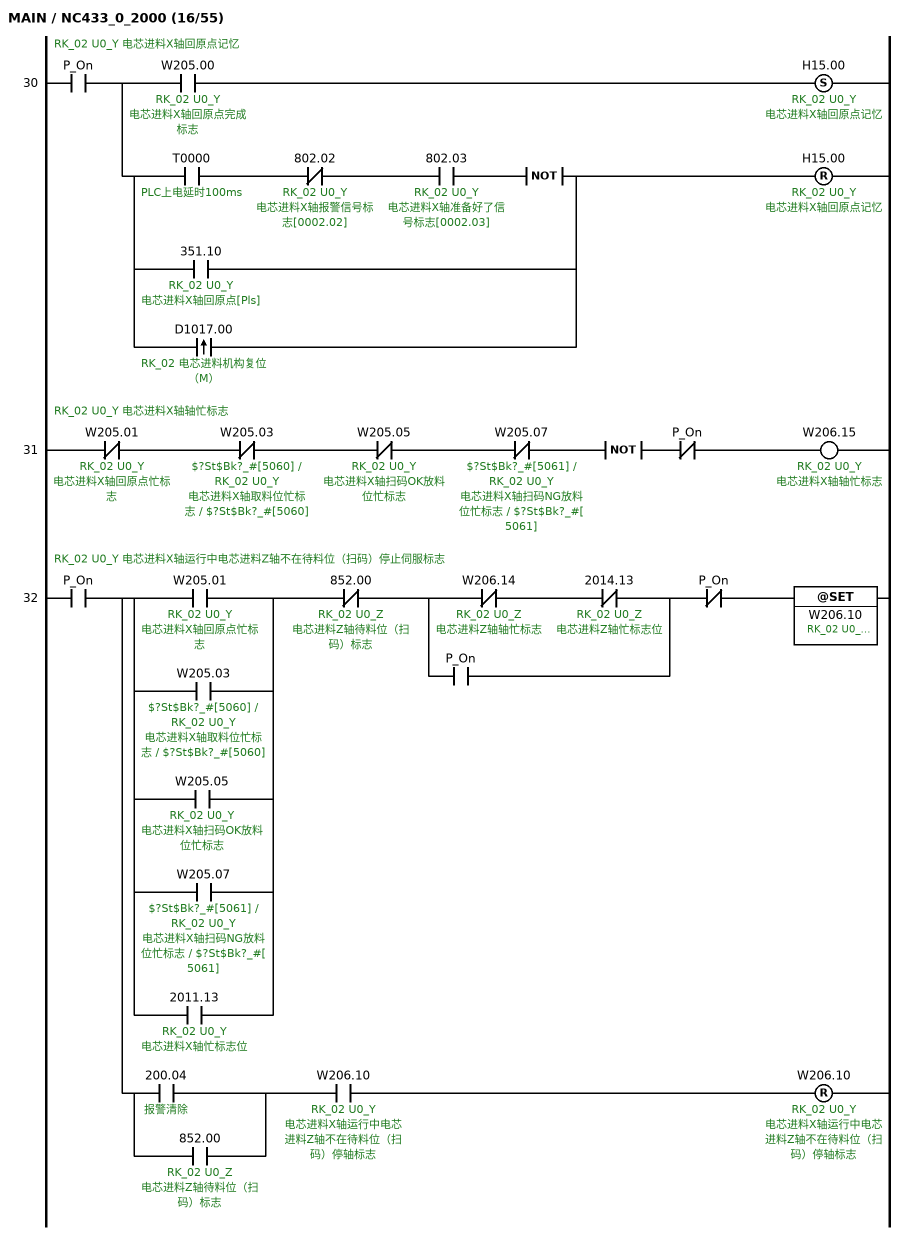
; rung 30: RK_02 U0_Y 电芯进料X轴回原点记忆
LD P_On
OUT TR0
AND W205.00  ; RK_02 U0_Y 电芯进料X轴回原点完成标志
SET H15.00  ; RK_02 U0_Y 电芯进料X轴回原点记忆
LD TR0
LD T0000  ; PLC上电延时100ms
ANDNOT 802.02  ; RK_02 U0_Y 电芯进料X轴报警信号标志[0002.02]
AND 802.03  ; RK_02 U0_Y 电芯进料X轴准备好了信号标志[0002.03]
NOT(520)
OR 351.10  ; RK_02 U0_Y 电芯进料X轴回原点[Pls]
@OR D1017.00  ; RK_02 电芯进料机构复位（M）
ANDLD
RSET H15.00  ; RK_02 U0_Y 电芯进料X轴回原点记忆
; rung 31: RK_02 U0_Y 电芯进料X轴轴忙标志
LDNOT W205.01  ; RK_02 U0_Y 电芯进料X轴回原点忙标志
ANDNOT W205.03  ; $?St$Bk?_#[5060] / RK_02 U0_Y 电芯进料X轴取料位忙标志 / $?St$Bk?_#[5060]
ANDNOT W205.05  ; RK_02 U0_Y 电芯进料X轴扫码OK放料位忙标志
ANDNOT W205.07  ; $?St$Bk?_#[5061] / RK_02 U0_Y 电芯进料X轴扫码NG放料位忙标志 / $?St$Bk?_#[5061]
NOT(520)
ANDNOT P_On
OUT W206.15  ; RK_02 U0_Y 电芯进料X轴轴忙标志
; rung 32: RK_02 U0_Y 电芯进料X轴运行中电芯进料Z轴不在待料位（扫码）停止伺服标志
LD P_On
OUT TR0
LD W205.01  ; RK_02 U0_Y 电芯进料X轴回原点忙标志
OR W205.03  ; $?St$Bk?_#[5060] / RK_02 U0_Y 电芯进料X轴取料位忙标志 / $?St$Bk?_#[5060]
OR W205.05  ; RK_02 U0_Y 电芯进料X轴扫码OK放料位忙标志
OR W205.07  ; $?St$Bk?_#[5061] / RK_02 U0_Y 电芯进料X轴扫码NG放料位忙标志 / $?St$Bk?_#[5061]
OR 2011.13  ; RK_02 U0_Y 电芯进料X轴忙标志位
ANDLD
ANDNOT 852.00  ; RK_02 U0_Z 电芯进料Z轴待料位（扫码）标志
LDNOT W206.14  ; RK_02 U0_Z 电芯进料Z轴轴忙标志
ANDNOT 2014.13  ; RK_02 U0_Z 电芯进料Z轴忙标志位
OR P_On
ANDLD
ANDNOT P_On
@SET W206.10  ; RK_02 U0_Y 电芯进料X轴运行中电芯进料Z轴不在待料位（扫码）停轴标志  // 增加相应报警信息
LD TR0
LD 200.04  ; 报警清除
OR 852.00  ; RK_02 U0_Z 电芯进料Z轴待料位（扫码）标志
ANDLD
AND W206.10  ; RK_02 U0_Y 电芯进料X轴运行中电芯进料Z轴不在待料位（扫码）停轴标志
RSET W206.10  ; RK_02 U0_Y 电芯进料X轴运行中电芯进料Z轴不在待料位（扫码）停轴标志

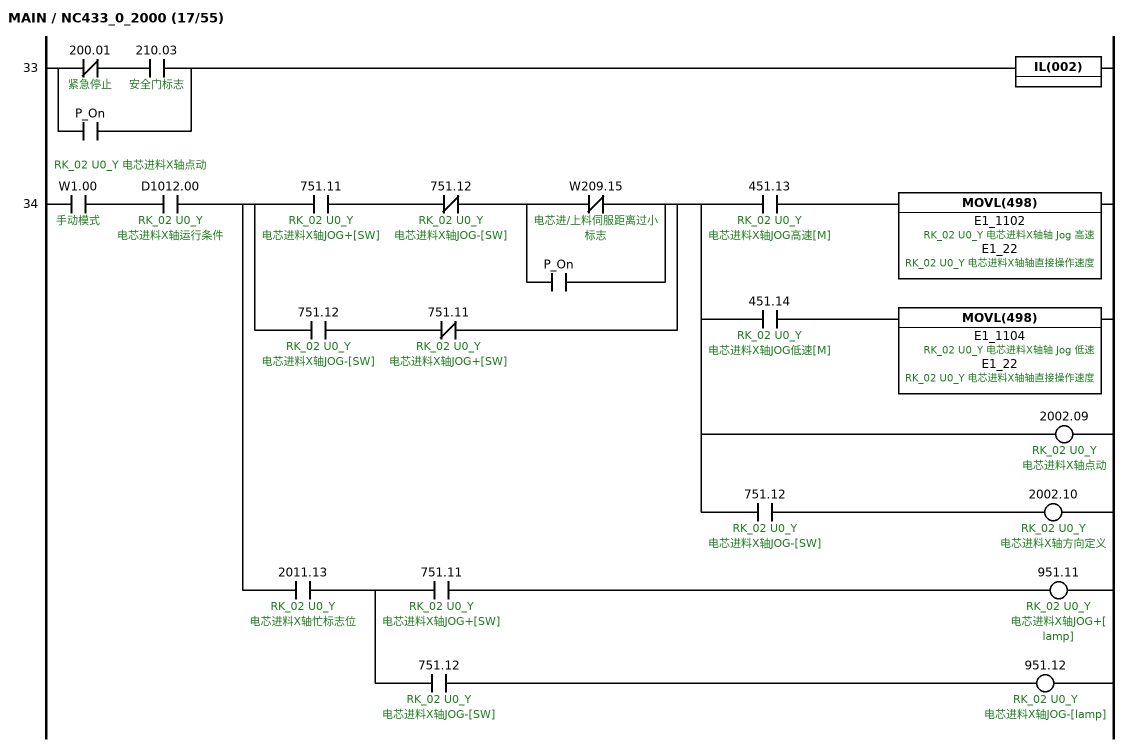
; rung 33
LDNOT 200.01  ; 紧急停止
AND 210.03  ; 安全门标志
OR P_On
IL(002)
; rung 34: RK_02 U0_Y 电芯进料X轴点动
LD W1.00  ; 手动模式
AND D1012.00  ; RK_02 U0_Y 电芯进料X轴运行条件
OUT TR0
LD 751.11  ; RK_02 U0_Y 电芯进料X轴JOG+[SW]
ANDNOT 751.12  ; RK_02 U0_Y 电芯进料X轴JOG-[SW]
LDNOT W209.15  ; 电芯进/上料伺服距离过小标志
OR P_On
ANDLD
LD 751.12  ; RK_02 U0_Y 电芯进料X轴JOG-[SW]
ANDNOT 751.11  ; RK_02 U0_Y 电芯进料X轴JOG+[SW]
ORLD
ANDLD
OUT TR1
AND 451.13  ; RK_02 U0_Y 电芯进料X轴JOG高速[M]
MOVL(498) E1_1102 E1_22  ; RK_02 U0_Y 电芯进料X轴轴 Jog 高速, RK_02 U0_Y 电芯进料X轴轴直接操作速度
LD TR1
AND 451.14  ; RK_02 U0_Y 电芯进料X轴JOG低速[M]
MOVL(498) E1_1104 E1_22  ; RK_02 U0_Y 电芯进料X轴轴 Jog 低速, RK_02 U0_Y 电芯进料X轴轴直接操作速度
LD TR1
OUT 2002.09  ; RK_02 U0_Y 电芯进料X轴点动
AND 751.12  ; RK_02 U0_Y 电芯进料X轴JOG-[SW]
OUT 2002.10  ; RK_02 U0_Y 电芯进料X轴方向定义
LD TR0
AND 2011.13  ; RK_02 U0_Y 电芯进料X轴忙标志位
OUT TR0
AND 751.11  ; RK_02 U0_Y 电芯进料X轴JOG+[SW]
OUT 951.11  ; RK_02 U0_Y 电芯进料X轴JOG+[lamp]
LD TR0
AND 751.12  ; RK_02 U0_Y 电芯进料X轴JOG-[SW]
OUT 951.12  ; RK_02 U0_Y 电芯进料X轴JOG-[lamp]

